  MoveC 565 to (267.87, -55.94, -4.17) mm, rotated rx -180 ry 0 rz -179 deg; joints [20.182, -52.388, 86.98, 32.921, -39.405, -26.577] to (267.42, -56.12, -4.17) mm, rotated rx -180 ry 0 rz -179 deg; joints [20.193, -52.411, 87.018, 32.927, -39.423, -26.576]
  MoveL 566 to (266.79, -56.12, -4.17) mm, rotated rx 180 ry 0 rz -179 deg; joints [20.201, -52.449, 87.082, 32.92, -39.448, -26.562]
  MoveC 567 to (266.34, -56.12, -3.99) mm, rotated rx -180 ry 0 rz -179 deg; joints [20.206, -52.481, 87.122, 32.922, -39.457, -26.561] to (266.15, -56.12, -3.54) mm, rotated rx -180 ry 0 rz -179 deg; joints [20.208, -52.505, 87.128, 32.937, -39.444, -26.579]
  Set speed (500.0 mm/s)
  MoveL 568 to (266.15, -56.12, 5) mm, rotated rx 180 ry 0 rz -179 deg; joints [20.208, -52.749, 86.893, 33.257, -39.042, -26.992]
  MoveL 569 to (266.15, -54.85, 5) mm, rotated rx -180 ry 0 rz -179 deg; joints [20.166, -52.775, 86.937, 33.185, -39.038, -26.93]
  Set speed (25.4 mm/s)
  MoveL 570 to (266.15, -54.85, 1.83) mm, rotated rx -180 ry 0 rz -179 deg; joints [20.166, -52.685, 87.025, 33.065, -39.187, -26.776]
  MoveL 571 to (266.15, -54.85, -7.71) mm, rotated rx -180 ry 0 rz -179 deg; joints [20.166, -52.411, 87.285, 32.712, -39.636, -26.319]
  MoveC 572 to (266.34, -54.85, -8.16) mm, rotated rx -180 ry 0 rz -179 deg; joints [20.164, -52.386, 87.279, 32.698, -39.65, -26.301] to (266.79, -54.85, -8.35) mm, rotated rx -180 ry 0 rz -179 deg; joints [20.158, -52.354, 87.239, 32.696, -39.641, -26.302]
  Set speed (50.8 mm/s)
  MoveL 573 to (267.42, -54.85, -8.35) mm, rotated rx 180 ry 0 rz -179 deg; joints [20.151, -52.317, 87.175, 32.702, -39.616, -26.316]
  MoveC 574 to (267.87, -55.04, -8.35) mm, rotated rx -180 ry 0 rz -179 deg; joints [20.152, -52.286, 87.124, 32.717, -39.599, -26.335] to (268.06, -55.49, -8.35) mm, rotated rx 180 ry 0 rz -179 deg; joints [20.165, -52.266, 87.09, 32.744, -39.593, -26.361]
  MoveL 575 to (268.06, -80.89, -8.35) mm, rotated rx -180 ry 0 rz -179 deg; joints [21.006, -51.73, 86.183, 34.166, -39.665, -27.586]
  MoveL 576 to (217.26, -80.89, -8.35) mm, rotated rx -180 ry 0 rz -179 deg; joints [21.633, -54.688, 91.144, 33.721, -41.611, -26.521]
  MoveL 577 to (217.26, -30.09, -8.35) mm, rotated rx -180 ry 0 rz -179 deg; joints [19.898, -55.732, 92.869, 30.944, -41.444, -24.2]
  MoveL 578 to (268.06, -30.09, -8.35) mm, rotated rx 180 ry 0 rz -179 deg; joints [19.315, -52.777, 87.951, 31.318, -39.52, -25.143]
  MoveL 579 to (268.06, -55.49, -8.35) mm, rotated rx 180 ry 0 rz -179 deg; joints [20.165, -52.266, 87.09, 32.744, -39.593, -26.361]
  MoveC 580 to (267.87, -55.94, -8.35) mm, rotated rx -180 ry 0 rz -179 deg; joints [20.182, -52.268, 87.093, 32.768, -39.601, -26.378] to (267.42, -56.12, -8.35) mm, rotated rx -180 ry 0 rz -179 deg; joints [20.193, -52.291, 87.131, 32.773, -39.62, -26.377]
  MoveL 581 to (266.79, -56.12, -8.35) mm, rotated rx -180 ry 0 rz -179 deg; joints [20.201, -52.328, 87.195, 32.767, -39.645, -26.363]
  MoveC 582 to (266.34, -56.12, -8.16) mm, rotated rx -180 ry 0 rz -179 deg; joints [20.206, -52.36, 87.235, 32.769, -39.654, -26.362] to (266.15, -56.12, -7.72) mm, rotated rx 180 ry 0 rz -179 deg; joints [20.208, -52.384, 87.241, 32.783, -39.64, -26.38]
  Set speed (500.0 mm/s)
  MoveL 583 to (266.15, -56.12, 6) mm, rotated rx -180 ry 0 rz -179 deg; joints [20.208, -52.777, 86.865, 33.295, -38.995, -27.041]
  MoveL 584 to (139.15, -54.85, 6) mm, rotated rx -180 ry 0 rz -179 deg; joints [21.754, -60.075, 98.759, 32.555, -43.53, -24.838]
  Set speed (25.4 mm/s)
  MoveL 585 to (139.15, -54.85, -3.54) mm, rotated rx 180 ry 0 rz -179 deg; joints [21.754, -59.764, 99.016, 32.238, -44.009, -24.398]
  MoveC 586 to (139.34, -54.85, -3.99) mm, rotated rx -180 ry 0 rz -179 deg; joints [21.751, -59.739, 99.012, 32.223, -44.026, -24.38] to (139.79, -54.85, -4.17) mm, rotated rx 180 ry 0 rz -179 deg; joints [21.745, -59.708, 98.977, 32.217, -44.02, -24.377]
  Set speed (50.8 mm/s)
  MoveL 587 to (140.42, -54.85, -4.17) mm, rotated rx -180 ry 0 rz -179 deg; joints [21.736, -59.673, 98.922, 32.217, -43.999, -24.385]
  MoveC 588 to (140.87, -55.04, -4.18) mm, rotated rx -180 ry 0 rz -179 deg; joints [21.737, -59.645, 98.876, 32.227, -43.985, -24.398] to (141.06, -55.49, -4.17) mm, rotated rx 180 ry 0 rz -179 deg; joints [21.75, -59.625, 98.845, 32.251, -43.981, -24.42]
  MoveL 589 to (141.06, -80.89, -4.17) mm, rotated rx 180 ry 0 rz -179 deg; joints [22.648, -59.084, 97.981, 33.603, -44.09, -25.514]
  MoveL 590 to (90.26, -80.89, -4.17) mm, rotated rx -180 ry 0 rz -179 deg; joints [23.379, -61.842, 102.338, 33.653, -45.731, -24.924]
  MoveL 591 to (90.26, -30.09, -4.17) mm, rotated rx -180 ry 0 rz -179 deg; joints [21.523, -62.92, 104.009, 30.966, -45.482, -22.818]
  MoveL 592 to (141.06, -30.09, -4.18) mm, rotated rx 180 ry 0 rz -179 deg; joints [20.842, -60.143, 99.667, 30.888, -43.873, -23.328]
  MoveL 593 to (141.06, -55.49, -4.17) mm, rotated rx 180 ry 0 rz -179 deg; joints [21.75, -59.625, 98.845, 32.251, -43.981, -24.42]
  MoveC 594 to (140.87, -55.94, -4.17) mm, rotated rx -180 ry 0 rz -179 deg; joints [21.769, -59.626, 98.847, 32.275, -43.989, -24.437] to (140.42, -56.12, -4.17) mm, rotated rx -180 ry 0 rz -179 deg; joints [21.782, -59.647, 98.88, 32.285, -44.005, -24.439]
  MoveL 595 to (139.79, -56.12, -4.18) mm, rotated rx -180 ry 0 rz -179 deg; joints [21.79, -59.682, 98.935, 32.285, -44.026, -24.431]
  MoveC 596 to (139.34, -56.12, -3.99) mm, rotated rx 180 ry 0 rz -179 deg; joints [21.796, -59.713, 98.97, 32.291, -44.031, -24.434] to (139.15, -56.12, -3.54) mm, rotated rx -180 ry 0 rz -179 deg; joints [21.799, -59.738, 98.974, 32.305, -44.015, -24.453]
  Set speed (500.0 mm/s)
  MoveL 597 to (139.15, -56.12, 5) mm, rotated rx -180 ry 0 rz -179 deg; joints [21.799, -60.016, 98.744, 32.59, -43.586, -24.847]
  MoveL 598 to (139.15, -54.85, 5) mm, rotated rx -180 ry 0 rz -179 deg; joints [21.754, -60.043, 98.786, 32.522, -43.58, -24.792]
  Set speed (25.4 mm/s)
  MoveL 599 to (139.15, -54.85, 1.83) mm, rotated rx -180 ry 0 rz -179 deg; joints [21.754, -59.94, 98.873, 32.415, -43.74, -24.644]
  MoveL 600 to (139.15, -54.85, -7.72) mm, rotated rx -180 ry 0 rz -179 deg; joints [21.754, -59.626, 99.126, 32.101, -44.219, -24.208]
  MoveC 601 to (139.34, -54.85, -8.16) mm, rotated rx -180 ry 0 rz -179 deg; joints [21.751, -59.601, 99.122, 32.087, -44.236, -24.19] to (139.79, -54.85, -8.35) mm, rotated rx -180 ry 0 rz -179 deg; joints [21.745, -59.57, 99.087, 32.081, -44.23, -24.187]
  Set speed (50.8 mm/s)
  MoveL 602 to (140.42, -54.85, -8.35) mm, rotated rx 180 ry 0 rz -179 deg; joints [21.736, -59.535, 99.032, 32.081, -44.209, -24.195]
  MoveC 603 to (140.87, -55.04, -8.35) mm, rotated rx 180 ry 0 rz -179 deg; joints [21.737, -59.507, 98.986, 32.091, -44.195, -24.209] to (141.06, -55.49, -8.35) mm, rotated rx 180 ry 0 rz -179 deg; joints [21.75, -59.487, 98.955, 32.115, -44.191, -24.23]
  MoveL 604 to (141.06, -80.89, -8.35) mm, rotated rx 180 ry 0 rz -179 deg; joints [22.648, -58.947, 98.091, 33.463, -44.295, -25.318]
  MoveL 605 to (90.26, -80.89, -8.35) mm, rotated rx -180 ry 0 rz -179 deg; joints [23.379, -61.699, 102.448, 33.516, -45.942, -24.728]
  MoveL 606 to (90.26, -30.09, -8.35) mm, rotated rx -180 ry 0 rz -179 deg; joints [21.523, -62.774, 104.119, 30.837, -45.702, -22.634]
  MoveL 607 to (141.06, -30.09, -8.35) mm, rotated rx 180 ry 0 rz -179 deg; joints [20.842, -60.004, 99.777, 30.756, -44.086, -23.144]
  MoveL 608 to (141.06, -55.49, -8.35) mm, rotated rx 180 ry 0 rz -179 deg; joints [21.75, -59.487, 98.955, 32.115, -44.191, -24.23]
  MoveC 609 to (140.87, -55.94, -8.35) mm, rotated rx 180 ry 0 rz -179 deg; joints [21.769, -59.488, 98.956, 32.139, -44.199, -24.247] to (140.42, -56.12, -8.35) mm, rotated rx 180 ry 0 rz -179 deg; joints [21.782, -59.509, 98.99, 32.149, -44.214, -24.249]
  MoveL 610 to (139.79, -56.12, -8.35) mm, rotated rx -180 ry 0 rz -179 deg; joints [21.79, -59.544, 99.045, 32.149, -44.235, -24.242]
  MoveC 611 to (139.34, -56.12, -8.16) mm, rotated rx -180 ry 0 rz -179 deg; joints [21.796, -59.575, 99.08, 32.155, -44.241, -24.245] to (139.15, -56.12, -7.72) mm, rotated rx -180 ry 0 rz -179 deg; joints [21.799, -59.6, 99.084, 32.169, -44.225, -24.263]
  Set speed (500.0 mm/s)
  MoveL 612 to (139.15, -56.12, 6) mm, rotated rx -180 ry 0 rz -179 deg; joints [21.799, -60.049, 98.717, 32.624, -43.536, -24.893]
  MoveL 613 to (139.15, -235.88, 6) mm, rotated rx -180 ry 0 rz -179 deg; joints [27.912, -55.671, 91.665, 42.031, -44.36, -32.8]
  Set speed (25.4 mm/s)
  MoveL 614 to (139.15, -235.88, -3.54) mm, rotated rx -180 ry 0 rz -179 deg; joints [27.912, -55.384, 91.924, 41.661, -44.767, -32.28]
  MoveC 615 to (139.34, -235.88, -3.99) mm, rotated rx -180 ry 0 rz -179 deg; joints [27.909, -55.36, 91.92, 41.644, -44.78, -32.26] to (139.79, -235.88, -4.17) mm, rotated rx 180 ry 0 rz -179 deg; joints [27.902, -55.33, 91.885, 41.639, -44.772, -32.258]
  Set speed (50.8 mm/s)
  MoveL 616 to (140.42, -235.89, -4.17) mm, rotated rx -180 ry 0 rz -179 deg; joints [27.891, -55.296, 91.828, 41.641, -44.75, -32.27]
  MoveC 617 to (140.87, -236.07, -4.18) mm, rotated rx 180 ry 0 rz -179 deg; joints [27.89, -55.266, 91.779, 41.653, -44.735, -32.287] to (141.06, -236.52, -4.17) mm, rotated rx 180 ry 0 rz -179 deg; joints [27.901, -55.244, 91.742, 41.676, -44.73, -32.311]
  MoveL 618 to (141.06, -261.92, -4.17) mm, rotated rx -180 ry 0 rz -179 deg; joints [28.717, -54.531, 90.562, 42.965, -44.828, -33.447]
  MoveL 619 to (90.26, -261.92, -4.17) mm, rotated rx 180 ry 0 rz -179 deg; joints [29.592, -57.246, 95.019, 42.834, -46.58, -32.507]
  MoveL 620 to (90.26, -211.12, -4.17) mm, rotated rx -180 ry 0 rz -179 deg; joints [27.914, -58.655, 97.294, 40.313, -46.353, -30.353]
  MoveL 621 to (141.06, -211.12, -4.17) mm, rotated rx -180 ry 0 rz -179 deg; joints [27.074, -55.932, 92.875, 40.38, -44.63, -31.184]
  MoveL 622 to (141.06, -236.52, -4.17) mm, rotated rx -180 ry 0 rz -179 deg; joints [27.901, -55.244, 91.742, 41.676, -44.73, -32.311]
  MoveC 623 to (140.87, -236.97, -4.18) mm, rotated rx -180 ry 0 rz -179 deg; joints [27.919, -55.241, 91.738, 41.698, -44.738, -32.327] to (140.42, -237.15, -4.18) mm, rotated rx 180 ry 0 rz -179 deg; joints [27.932, -55.261, 91.77, 41.706, -44.755, -32.327]
  MoveL 624 to (139.79, -237.15, -4.18) mm, rotated rx -180 ry 0 rz -179 deg; joints [27.943, -55.295, 91.827, 41.703, -44.777, -32.315]
  MoveC 625 to (139.34, -237.16, -3.99) mm, rotated rx -180 ry 0 rz -179 deg; joints [27.95, -55.325, 91.862, 41.709, -44.785, -32.316] to (139.15, -237.15, -3.54) mm, rotated rx -180 ry 0 rz -179 deg; joints [27.953, -55.349, 91.867, 41.725, -44.772, -32.337]
  Set speed (500.0 mm/s)
  MoveL 626 to (139.15, -237.15, 5) mm, rotated rx -180 ry 0 rz -179 deg; joints [27.953, -55.606, 91.635, 42.057, -44.408, -32.802]
  MoveL 627 to (139.15, -235.88, 5) mm, rotated rx -180 ry 0 rz -179 deg; joints [27.912, -55.641, 91.693, 41.992, -44.403, -32.745]
  Set speed (25.4 mm/s)
  MoveL 628 to (139.15, -235.88, 1.83) mm, rotated rx -180 ry 0 rz -179 deg; joints [27.912, -55.546, 91.779, 41.868, -44.538, -32.571]
  MoveL 629 to (139.15, -235.88, -7.72) mm, rotated rx 180 ry 0 rz -179 deg; joints [27.912, -55.257, 92.036, 41.502, -44.946, -32.056]
  MoveC 630 to (139.34, -235.88, -8.16) mm, rotated rx -180 ry 0 rz -179 deg; joints [27.909, -55.233, 92.031, 41.485, -44.959, -32.035] to (139.79, -235.88, -8.35) mm, rotated rx 180 ry 0 rz -179 deg; joints [27.902, -55.203, 91.996, 41.48, -44.951, -32.034]
  Set speed (50.8 mm/s)
  MoveL 631 to (140.42, -235.89, -8.35) mm, rotated rx -180 ry 0 rz -179 deg; joints [27.891, -55.168, 91.939, 41.482, -44.928, -32.046]
  MoveC 632 to (140.87, -236.07, -8.35) mm, rotated rx -180 ry 0 rz -179 deg; joints [27.89, -55.139, 91.89, 41.493, -44.913, -32.063] to (141.06, -236.52, -8.35) mm, rotated rx -180 ry 0 rz -179 deg; joints [27.901, -55.116, 91.853, 41.517, -44.908, -32.087]
  MoveL 633 to (141.06, -261.92, -8.35) mm, rotated rx -180 ry 0 rz -179 deg; joints [28.717, -54.405, 90.673, 42.803, -45.001, -33.219]
  MoveL 634 to (90.26, -261.92, -8.35) mm, rotated rx -180 ry 0 rz -179 deg; joints [29.592, -57.114, 95.129, 42.679, -46.758, -32.28]
  MoveL 635 to (90.26, -211.12, -8.35) mm, rotated rx -180 ry 0 rz -179 deg; joints [27.914, -58.519, 97.404, 40.162, -46.54, -30.135]
  MoveL 636 to (141.06, -211.12, -8.35) mm, rotated rx -180 ry 0 rz -179 deg; joints [27.074, -55.803, 92.986, 40.224, -44.813, -30.964]
  MoveL 637 to (141.06, -236.52, -8.35) mm, rotated rx -180 ry 0 rz -179 deg; joints [27.901, -55.116, 91.853, 41.517, -44.908, -32.087]
  MoveC 638 to (140.87, -236.97, -8.35) mm, rotated rx -180 ry 0 rz -179 deg; joints [27.919, -55.114, 91.849, 41.539, -44.916, -32.103] to (140.42, -237.16, -8.35) mm, rotated rx -180 ry 0 rz -179 deg; joints [27.932, -55.133, 91.881, 41.547, -44.933, -32.102]
  MoveL 639 to (139.79, -237.16, -8.35) mm, rotated rx -180 ry 0 rz -179 deg; joints [27.943, -55.168, 91.938, 41.544, -44.955, -32.09]
  MoveC 640 to (139.34, -237.15, -8.16) mm, rotated rx 180 ry 0 rz -179 deg; joints [27.95, -55.198, 91.973, 41.55, -44.963, -32.091] to (139.15, -237.15, -7.72) mm, rotated rx -180 ry 0 rz -179 deg; joints [27.953, -55.222, 91.978, 41.566, -44.951, -32.112]
  Set speed (500.0 mm/s)
  MoveL 641 to (139.15, -237.15, 6) mm, rotated rx -180 ry 0 rz -179 deg; joints [27.953, -55.636, 91.607, 42.096, -44.366, -32.857]
  MoveL 642 to (266.15, -235.88, 6) mm, rotated rx -180 ry 0 rz -179 deg; joints [25.965, -48.371, 79.367, 43.399, -39.586, -36.084]
  Set speed (25.4 mm/s)
  MoveL 643 to (266.15, -235.89, -3.54) mm, rotated rx -180 ry 0 rz -179 deg; joints [25.965, -48.122, 79.642, 42.969, -39.967, -35.524]
  MoveC 644 to (266.34, -235.88, -3.99) mm, rotated rx -180 ry 0 rz -179 deg; joints [25.963, -48.099, 79.635, 42.953, -39.977, -35.504] to (266.79, -235.89, -4.17) mm, rotated rx -180 ry 0 rz -179 deg; joints [25.956, -48.067, 79.593, 42.953, -39.966, -35.509]
  Set speed (50.8 mm/s)
  MoveL 645 to (267.42, -235.89, -4.18) mm, rotated rx -180 ry 0 rz -179 deg; joints [25.947, -48.029, 79.526, 42.964, -39.94, -35.53]
  MoveC 646 to (267.87, -236.07, -4.17) mm, rotated rx 180 ry 0 rz -179 deg; joints [25.947, -47.996, 79.47, 42.983, -39.923, -35.554] to (268.06, -236.52, -4.18) mm, rotated rx -180 ry 0 rz -179 deg; joints [25.958, -47.972, 79.428, 43.011, -39.916, -35.584]
  MoveL 647 to (268.06, -261.92, -4.18) mm, rotated rx 180 ry 0 rz -179 deg; joints [26.731, -47.239, 78.154, 44.43, -39.983, -36.912]
  MoveL 648 to (217.26, -261.92, -4.18) mm, rotated rx -180 ry 0 rz -179 deg; joints [27.493, -50.26, 83.367, 43.615, -42.008, -35.297]
  MoveL 649 to (217.26, -211.12, -4.17) mm, rotated rx -180 ry 0 rz -179 deg; joints [25.902, -51.672, 85.769, 40.9, -41.85, -32.832]
  MoveL 650 to (268.06, -211.12, -4.17) mm, rotated rx 180 ry 0 rz -179 deg; joints [25.174, -48.676, 80.646, 41.595, -39.848, -34.275]
  MoveL 651 to (268.06, -236.52, -4.18) mm, rotated rx -180 ry 0 rz -179 deg; joints [25.958, -47.972, 79.428, 43.011, -39.916, -35.584]
  MoveC 652 to (267.87, -236.97, -4.17) mm, rotated rx -180 ry 0 rz -179 deg; joints [25.974, -47.971, 79.426, 43.033, -39.925, -35.601] to (267.42, -237.16, -4.18) mm, rotated rx 180 ry 0 rz -179 deg; joints [25.986, -47.993, 79.464, 43.035, -39.944, -35.596]
  MoveL 653 to (266.79, -237.15, -4.17) mm, rotated rx -180 ry 0 rz -179 deg; joints [25.995, -48.031, 79.531, 43.023, -39.97, -35.574]
  MoveC 654 to (266.34, -237.15, -3.99) mm, rotated rx 180 ry 0 rz -179 deg; joints [26.002, -48.063, 79.573, 43.024, -39.981, -35.57] to (266.15, -237.16, -3.54) mm, rotated rx -180 ry 0 rz -179 deg; joints [26.004, -48.087, 79.579, 43.04, -39.97, -35.59]
  Set speed (500.0 mm/s)
  MoveL 655 to (266.15, -237.15, 5) mm, rotated rx 180 ry 0 rz -179 deg; joints [26.004, -48.309, 79.334, 43.425, -39.629, -36.091]
  MoveL 656 to (266.15, -235.89, 5) mm, rotated rx -180 ry 0 rz -179 deg; joints [25.965, -48.345, 79.397, 43.354, -39.626, -36.024]
  Set speed (25.4 mm/s)
  MoveL 657 to (266.15, -235.88, 1.83) mm, rotated rx 180 ry 0 rz -179 deg; joints [25.965, -48.263, 79.488, 43.21, -39.752, -35.837]
  MoveL 658 to (266.15, -235.89, -7.71) mm, rotated rx -180 ry 0 rz -179 deg; joints [25.965, -48.012, 79.759, 42.785, -40.134, -35.283]
  MoveC 659 to (266.34, -235.88, -8.16) mm, rotated rx 180 ry 0 rz -179 deg; joints [25.963, -47.989, 79.752, 42.769, -40.144, -35.264] to (266.79, -235.89, -8.35) mm, rotated rx -180 ry 0 rz -179 deg; joints [25.956, -47.957, 79.71, 42.768, -40.133, -35.268]
  Set speed (50.8 mm/s)
  MoveL 660 to (267.42, -235.89, -8.35) mm, rotated rx -180 ry 0 rz -179 deg; joints [25.947, -47.918, 79.643, 42.78, -40.107, -35.289]
  MoveC 661 to (267.87, -236.07, -8.35) mm, rotated rx -180 ry 0 rz -179 deg; joints [25.947, -47.886, 79.587, 42.798, -40.089, -35.313] to (268.06, -236.52, -8.35) mm, rotated rx -180 ry 0 rz -179 deg; joints [25.958, -47.862, 79.545, 42.826, -40.083, -35.343]
  MoveL 662 to (268.06, -261.92, -8.35) mm, rotated rx -180 ry 0 rz -179 deg; joints [26.731, -47.13, 78.272, 44.241, -40.145, -36.665]
  MoveL 663 to (217.26, -261.92, -8.35) mm, rotated rx -180 ry 0 rz -179 deg; joints [27.493, -50.144, 83.481, 43.439, -42.175, -35.06]
  MoveL 664 to (217.26, -211.12, -8.35) mm, rotated rx -180 ry 0 rz -179 deg; joints [25.902, -51.553, 85.883, 40.731, -42.026, -32.605]
  MoveL 665 to (268.06, -211.12, -8.35) mm, rotated rx 180 ry 0 rz -179 deg; joints [25.174, -48.564, 80.762, 41.414, -40.019, -34.04]
  MoveL 666 to (268.06, -236.52, -8.35) mm, rotated rx -180 ry 0 rz -179 deg; joints [25.958, -47.862, 79.545, 42.826, -40.083, -35.343]
  MoveC 667 to (267.87, -236.97, -8.35) mm, rotated rx -180 ry 0 rz -179 deg; joints [25.974, -47.86, 79.543, 42.848, -40.092, -35.36] to (267.42, -237.16, -8.35) mm, rotated rx -180 ry 0 rz -179 deg; joints [25.986, -47.882, 79.581, 42.85, -40.11, -35.354]
  MoveL 668 to (266.79, -237.15, -8.35) mm, rotated rx -180 ry 0 rz -179 deg; joints [25.995, -47.921, 79.648, 42.839, -40.136, -35.333]
  MoveC 669 to (266.34, -237.15, -8.16) mm, rotated rx 180 ry 0 rz -179 deg; joints [26.002, -47.953, 79.69, 42.839, -40.147, -35.329] to (266.15, -237.16, -7.72) mm, rotated rx -180 ry 0 rz -179 deg; joints [26.004, -47.976, 79.697, 42.856, -40.137, -35.349]
  Set speed (500.0 mm/s)
  MoveL 670 to (266.15, -237.16, 6) mm, rotated rx -180 ry 0 rz -179 deg; joints [26.004, -48.335, 79.305, 43.471, -39.59, -36.15]
  MoveL 671 to (393.15, -235.88, 6) mm, rotated rx -180 ry 0 rz -179 deg; joints [24.267, -39.923, 64.425, 47.387, -33.948, -42.041]
  Set speed (25.4 mm/s)
  MoveL 672 to (393.15, -235.88, -3.54) mm, rotated rx -180 ry 0 rz -179 deg; joints [24.267, -39.722, 64.741, 46.829, -34.299, -41.367]
  MoveC 673 to (393.34, -235.88, -3.99) mm, rotated rx 180 ry 0 rz -179 deg; joints [24.264, -39.699, 64.731, 46.812, -34.307, -41.348] to (393.79, -235.89, -4.17) mm, rotated rx -180 ry 0 rz -179 deg; joints [24.259, -39.662, 64.677, 46.822, -34.292, -41.363]
  Set speed (50.8 mm/s)
  MoveL 674 to (394.42, -235.88, -4.18) mm, rotated rx 180 ry 0 rz -179 deg; joints [24.251, -39.615, 64.592, 46.852, -34.26, -41.404]
  MoveC 675 to (394.87, -236.07, -4.18) mm, rotated rx -180 ry 0 rz -179 deg; joints [24.25, -39.576, 64.522, 46.886, -34.239, -41.445] to (395.06, -236.52, -4.17) mm, rotated rx -180 ry 0 rz -179 deg; joints [24.261, -39.549, 64.471, 46.925, -34.23, -41.486]
  MoveL 676 to (395.06, -261.92, -4.18) mm, rotated rx -180 ry 0 rz -179 deg; joints [24.996, -38.724, 62.973, 48.623, -34.272, -43.171]
  MoveL 677 to (344.26, -261.92, -4.18) mm, rotated rx 180 ry 0 rz -179 deg; joints [25.663, -42.34, 69.501, 46.465, -36.682, -40.167]
  MoveL 678 to (344.26, -211.12, -4.17) mm, rotated rx -180 ry 0 rz -179 deg; joints [24.154, -43.854, 72.2, 43.366, -36.579, -37.18]
  MoveL 679 to (395.06, -211.12, -4.18) mm, rotated rx 180 ry 0 rz -179 deg; joints [23.519, -40.332, 65.889, 45.25, -34.187, -39.843]
  MoveL 680 to (395.06, -236.52, -4.17) mm, rotated rx -180 ry 0 rz -179 deg; joints [24.261, -39.549, 64.471, 46.925, -34.23, -41.486]
  MoveC 681 to (394.87, -236.97, -4.18) mm, rotated rx 180 ry 0 rz -179 deg; joints [24.277, -39.548, 64.47, 46.946, -34.24, -41.503] to (394.42, -237.16, -4.18) mm, rotated rx 180 ry 0 rz -179 deg; joints [24.288, -39.575, 64.52, 46.937, -34.263, -41.487]
  MoveL 682 to (393.79, -237.16, -4.17) mm, rotated rx -180 ry 0 rz -179 deg; joints [24.296, -39.622, 64.604, 46.907, -34.294, -41.446]
  MoveC 683 to (393.34, -237.15, -3.99) mm, rotated rx -180 ry 0 rz -179 deg; joints [24.301, -39.659, 64.658, 46.896, -34.309, -41.431] to (393.15, -237.16, -3.54) mm, rotated rx 180 ry 0 rz -179 deg; joints [24.304, -39.682, 64.668, 46.913, -34.302, -41.45]
  Set speed (500.0 mm/s)
  MoveL 684 to (393.15, -237.16, 5) mm, rotated rx -180 ry 0 rz -179 deg; joints [24.304, -39.862, 64.386, 47.412, -33.988, -42.054]
  MoveL 685 to (393.15, -235.88, 5) mm, rotated rx -180 ry 0 rz -179 deg; joints [24.267, -39.902, 64.459, 47.328, -33.985, -41.97]
  Set speed (25.4 mm/s)
  MoveL 686 to (393.15, -235.88, 1.82) mm, rotated rx 180 ry 0 rz -179 deg; joints [24.267, -39.836, 64.565, 47.141, -34.102, -41.744]
  MoveL 687 to (393.15, -235.88, -7.72) mm, rotated rx -180 ry 0 rz -179 deg; joints [24.267, -39.632, 64.875, 46.59, -34.453, -41.078]
  MoveC 688 to (393.34, -235.88, -8.16) mm, rotated rx 180 ry 0 rz -179 deg; joints [24.264, -39.609, 64.865, 46.573, -34.461, -41.059] to (393.79, -235.89, -8.35) mm, rotated rx 180 ry 0 rz -179 deg; joints [24.259, -39.572, 64.811, 46.584, -34.446, -41.074]
  Set speed (50.8 mm/s)
  MoveL 689 to (394.42, -235.89, -8.35) mm, rotated rx -180 ry 0 rz -179 deg; joints [24.251, -39.526, 64.727, 46.613, -34.414, -41.114]
  MoveC 690 to (394.87, -236.07, -8.35) mm, rotated rx -180 ry 0 rz -179 deg; joints [24.25, -39.487, 64.657, 46.647, -34.392, -41.155] to (395.06, -236.52, -8.35) mm, rotated rx -180 ry 0 rz -179 deg; joints [24.261, -39.459, 64.606, 46.685, -34.384, -41.196]
  MoveL 691 to (395.06, -261.92, -8.35) mm, rotated rx -180 ry 0 rz -179 deg; joints [24.996, -38.637, 63.11, 48.377, -34.421, -42.872]
  MoveL 692 to (344.26, -261.92, -8.35) mm, rotated rx -180 ry 0 rz -179 deg; joints [25.663, -42.243, 69.629, 46.248, -36.837, -39.896]
  MoveL 693 to (344.26, -211.12, -8.35) mm, rotated rx 180 ry 0 rz -179 deg; joints [24.154, -43.753, 72.324, 43.159, -36.742, -36.922]
  MoveL 694 to (395.06, -211.12, -8.35) mm, rotated rx -180 ry 0 rz -179 deg; joints [23.519, -40.24, 66.022, 45.016, -34.345, -39.561]
  MoveL 695 to (395.06, -236.52, -8.35) mm, rotated rx -180 ry 0 rz -179 deg; joints [24.261, -39.459, 64.606, 46.685, -34.384, -41.196]
  MoveC 696 to (394.87, -236.97, -8.35) mm, rotated rx -180 ry 0 rz -179 deg; joints [24.277, -39.459, 64.605, 46.706, -34.394, -41.213] to (394.42, -237.16, -8.35) mm, rotated rx -180 ry 0 rz -179 deg; joints [24.288, -39.486, 64.654, 46.697, -34.416, -41.197]
  MoveL 697 to (393.79, -237.16, -8.35) mm, rotated rx -180 ry 0 rz -179 deg; joints [24.296, -39.532, 64.739, 46.667, -34.447, -41.157]
  MoveC 698 to (393.34, -237.15, -8.16) mm, rotated rx -180 ry 0 rz -179 deg; joints [24.301, -39.569, 64.793, 46.657, -34.463, -41.141] to (393.15, -237.16, -7.72) mm, rotated rx -180 ry 0 rz -179 deg; joints [24.304, -39.592, 64.803, 46.674, -34.455, -41.16]
  Set speed (500.0 mm/s)
  MoveL 699 to (393.15, -237.16, 6) mm, rotated rx -180 ry 0 rz -179 deg; joints [24.304, -39.882, 64.352, 47.472, -33.951, -42.125]
  MoveL 700 to (393.15, -422.22, 6) mm, rotated rx 180 ry 0 rz -179 deg; joints [29.464, -32.65, 51.048, 60.809, -34.294, -55.932]
  Set speed (25.4 mm/s)
  MoveL 701 to (393.15, -422.22, -3.54) mm, rotated rx -180 ry 0 rz -179 deg; joints [29.464, -32.503, 51.438, 60.128, -34.558, -55.107]
  MoveC 702 to (393.34, -422.22, -3.99) mm, rotated rx -180 ry 0 rz -179 deg; joints [29.462, -32.479, 51.425, 60.112, -34.562, -55.088] to (393.79, -422.22, -4.17) mm, rotated rx 180 ry 0 rz -179 deg; joints [29.455, -32.437, 51.358, 60.136, -34.544, -55.12]
  Set speed (50.8 mm/s)
  MoveL 703 to (394.42, -422.22, -4.18) mm, rotated rx 180 ry 0 rz -179 deg; joints [29.446, -32.38, 51.252, 60.189, -34.512, -55.187]
  MoveC 704 to (394.87, -422.41, -4.17) mm, rotated rx -180 ry 0 rz -179 deg; joints [29.445, -32.331, 51.161, 60.241, -34.49, -55.252] to (395.06, -422.86, -4.17) mm, rotated rx -180 ry 0 rz -179 deg; joints [29.454, -32.293, 51.089, 60.293, -34.481, -55.311]
  MoveL 705 to (395.06, -448.26, -4.17) mm, rotated rx -180 ry 0 rz -179 deg; joints [30.126, -31.02, 48.698, 62.376, -34.505, -57.583]
  MoveL 706 to (344.26, -448.26, -4.17) mm, rotated rx -180 ry 0 rz -179 deg; joints [30.888, -35.354, 56.786, 58.582, -36.981, -52.597]
  MoveL 707 to (344.26, -397.46, -4.17) mm, rotated rx -180 ry 0 rz -179 deg; joints [29.512, -37.525, 60.781, 55.102, -36.914, -48.897]
  MoveL 708 to (395.06, -397.46, -4.18) mm, rotated rx -180 ry 0 rz -179 deg; joints [28.773, -33.479, 53.306, 58.299, -34.454, -53.166]
  MoveL 709 to (395.06, -422.86, -4.17) mm, rotated rx -180 ry 0 rz -179 deg; joints [29.454, -32.293, 51.089, 60.293, -34.481, -55.311]
  MoveC 710 to (394.87, -423.31, -4.18) mm, rotated rx 180 ry 0 rz -179 deg; joints [29.469, -32.288, 51.08, 60.313, -34.491, -55.329] to (394.42, -423.49, -4.18) mm, rotated rx 180 ry 0 rz -179 deg; joints [29.48, -32.319, 51.138, 60.29, -34.513, -55.297]
  MoveL 711 to (393.79, -423.49, -4.18) mm, rotated rx -180 ry 0 rz -179 deg; joints [29.489, -32.376, 51.244, 60.237, -34.545, -55.23]
  MoveC 712 to (393.34, -423.49, -3.99) mm, rotated rx -180 ry 0 rz -179 deg; joints [29.496, -32.418, 51.311, 60.213, -34.563, -55.198] to (393.15, -423.49, -3.54) mm, rotated rx 180 ry 0 rz -179 deg; joints [29.498, -32.442, 51.324, 60.229, -34.56, -55.216]
  Set speed (500.0 mm/s)
  MoveL 713 to (393.15, -423.49, 5) mm, rotated rx -180 ry 0 rz -179 deg; joints [29.498, -32.573, 50.974, 60.839, -34.324, -55.955]
  MoveL 714 to (393.15, -422.22, 5) mm, rotated rx 180 ry 0 rz -179 deg; joints [29.464, -32.635, 51.09, 60.737, -34.322, -55.845]
  Set speed (25.4 mm/s)
  MoveL 715 to (393.15, -422.22, 1.82) mm, rotated rx -180 ry 0 rz -179 deg; joints [29.464, -32.586, 51.22, 60.509, -34.41, -55.568]
  MoveL 716 to (393.15, -422.22, -7.72) mm, rotated rx 180 ry 0 rz -179 deg; joints [29.464, -32.436, 51.604, 59.836, -34.675, -54.752]
  MoveC 717 to (393.34, -422.22, -8.16) mm, rotated rx 180 ry 0 rz -179 deg; joints [29.462, -32.413, 51.591, 59.82, -34.678, -54.734] to (393.79, -422.22, -8.35) mm, rotated rx -180 ry 0 rz -179 deg; joints [29.455, -32.37, 51.524, 59.844, -34.661, -54.765]
  Set speed (50.8 mm/s)
  MoveL 718 to (394.42, -422.22, -8.35) mm, rotated rx -180 ry 0 rz -179 deg; joints [29.446, -32.314, 51.419, 59.896, -34.629, -54.832]
  MoveC 719 to (394.87, -422.41, -8.35) mm, rotated rx -180 ry 0 rz -179 deg; joints [29.445, -32.265, 51.328, 59.948, -34.606, -54.896] to (395.06, -422.86, -8.35) mm, rotated rx -180 ry 0 rz -179 deg; joints [29.454, -32.227, 51.256, 59.999, -34.597, -54.954]
  MoveL 720 to (395.06, -448.26, -8.35) mm, rotated rx -180 ry 0 rz -179 deg; joints [30.126, -30.959, 48.874, 62.073, -34.615, -57.215]
  MoveL 721 to (344.26, -448.26, -8.35) mm, rotated rx 180 ry 0 rz -179 deg; joints [30.888, -35.277, 56.936, 58.325, -37.1, -52.274]
  MoveL 722 to (344.26, -397.46, -8.35) mm, rotated rx -180 ry 0 rz -179 deg; joints [29.512, -37.441, 60.923, 54.857, -37.043, -48.59]
  MoveL 723 to (395.06, -397.46, -8.35) mm, rotated rx 180 ry 0 rz -179 deg; joints [28.773, -33.409, 53.466, 58.014, -34.576, -52.82]
  MoveL 724 to (395.06, -422.86, -8.35) mm, rotated rx -180 ry 0 rz -179 deg; joints [29.454, -32.227, 51.256, 59.999, -34.597, -54.954]
  MoveC 725 to (394.87, -423.31, -8.35) mm, rotated rx 180 ry 0 rz -179 deg; joints [29.469, -32.222, 51.247, 60.019, -34.607, -54.973] to (394.42, -423.49, -8.35) mm, rotated rx -180 ry 0 rz -179 deg; joints [29.48, -32.253, 51.305, 59.997, -34.629, -54.941]
  MoveL 726 to (393.79, -423.49, -8.35) mm, rotated rx -180 ry 0 rz -179 deg; joints [29.489, -32.309, 51.41, 59.945, -34.662, -54.874]
  MoveC 727 to (393.34, -423.49, -8.16) mm, rotated rx 180 ry 0 rz -179 deg; joints [29.496, -32.352, 51.477, 59.921, -34.679, -54.842] to (393.15, -423.49, -7.72) mm, rotated rx 180 ry 0 rz -179 deg; joints [29.498, -32.376, 51.49, 59.937, -34.676, -54.861]
  Set speed (500.0 mm/s)
  MoveL 728 to (393.15, -423.49, 6) mm, rotated rx -180 ry 0 rz -179 deg; joints [29.498, -32.588, 50.933, 60.911, -34.296, -56.043]
  MoveL 729 to (266.15, -422.22, 6) mm, rotated rx 180 ry 0 rz -179 deg; joints [31.414, -42.203, 68.526, 54.019, -40.099, -46.494]
  Set speed (25.4 mm/s)
  MoveL 730 to (266.15, -422.22, -3.54) mm, rotated rx 180 ry 0 rz -179 deg; joints [31.414, -41.989, 68.827, 53.528, -40.404, -45.851]
  MoveC 731 to (266.34, -422.22, -3.99) mm, rotated rx -180 ry 0 rz -179 deg; joints [31.411, -41.966, 68.819, 53.511, -40.41, -45.83] to (266.79, -422.22, -4.17) mm, rotated rx -180 ry 0 rz -179 deg; joints [31.404, -41.933, 68.773, 53.515, -40.397, -45.84]
  Set speed (50.8 mm/s)
  MoveL 732 to (267.42, -422.22, -4.17) mm, rotated rx -180 ry 0 rz -179 deg; joints [31.394, -41.892, 68.698, 53.535, -40.37, -45.873]
  MoveC 733 to (267.87, -422.41, -4.18) mm, rotated rx -180 ry 0 rz -179 deg; joints [31.392, -41.855, 68.633, 53.56, -40.352, -45.907] to (268.06, -422.86, -4.18) mm, rotated rx -180 ry 0 rz -179 deg; joints [31.401, -41.826, 68.581, 53.592, -40.345, -45.943]
  MoveL 734 to (268.06, -448.26, -4.17) mm, rotated rx 180 ry 0 rz -179 deg; joints [32.101, -40.832, 66.792, 55.092, -40.391, -47.504]
  MoveL 735 to (217.26, -448.26, -4.17) mm, rotated rx -180 ry 0 rz -179 deg; joints [32.96, -44.063, 72.571, 53.644, -42.497, -45.048]
  MoveL 736 to (217.26, -397.46, -4.18) mm, rotated rx 180 ry 0 rz -179 deg; joints [31.527, -45.926, 75.859, 50.875, -42.38, -42.245]
  MoveL 737 to (268.06, -397.46, -4.18) mm, rotated rx -180 ry 0 rz -179 deg; joints [30.691, -42.778, 70.284, 52.113, -40.295, -44.428]
  MoveL 738 to (268.06, -422.86, -4.18) mm, rotated rx -180 ry 0 rz -179 deg; joints [31.401, -41.826, 68.581, 53.592, -40.345, -45.943]
  MoveC 739 to (267.87, -423.31, -4.17) mm, rotated rx -180 ry 0 rz -179 deg; joints [31.417, -41.821, 68.571, 53.613, -40.353, -45.961] to (267.42, -423.49, -4.17) mm, rotated rx -180 ry 0 rz -179 deg; joints [31.429, -41.843, 68.611, 53.61, -40.373, -45.949]
  MoveL 740 to (266.79, -423.49, -4.17) mm, rotated rx -180 ry 0 rz -179 deg; joints [31.439, -41.884, 68.685, 53.59, -40.4, -45.917]
  MoveC 741 to (266.34, -423.49, -3.99) mm, rotated rx -180 ry 0 rz -179 deg; joints [31.447, -41.918, 68.732, 53.585, -40.413, -45.907] to (266.15, -423.49, -3.54) mm, rotated rx -180 ry 0 rz -179 deg; joints [31.45, -41.94, 68.74, 53.602, -40.406, -45.927]
  Set speed (500.0 mm/s)
  MoveL 742 to (266.15, -423.49, 5) mm, rotated rx -180 ry 0 rz -179 deg; joints [31.45, -42.132, 68.471, 54.041, -40.134, -46.503]
  MoveL 743 to (266.15, -422.22, 5) mm, rotated rx 180 ry 0 rz -179 deg; joints [31.414, -42.181, 68.558, 53.967, -40.131, -46.426]
  Set speed (25.4 mm/s)
  MoveL 744 to (266.15, -422.22, 1.82) mm, rotated rx 180 ry 0 rz -179 deg; joints [31.414, -42.11, 68.659, 53.802, -40.233, -46.211]
  MoveL 745 to (266.15, -422.22, -7.71) mm, rotated rx -180 ry 0 rz -179 deg; joints [31.414, -41.893, 68.956, 53.317, -40.538, -45.573]
  MoveC 746 to (266.34, -422.22, -8.16) mm, rotated rx 180 ry 0 rz -179 deg; joints [31.411, -41.871, 68.948, 53.3, -40.544, -45.553] to (266.79, -422.22, -8.35) mm, rotated rx 180 ry 0 rz -179 deg; joints [31.404, -41.837, 68.901, 53.304, -40.531, -45.563]
  Set speed (50.8 mm/s)
  MoveL 747 to (267.42, -422.22, -8.35) mm, rotated rx -180 ry 0 rz -179 deg; joints [31.394, -41.796, 68.827, 53.324, -40.504, -45.595]
  MoveC 748 to (267.87, -422.41, -8.35) mm, rotated rx -180 ry 0 rz -179 deg; joints [31.392, -41.76, 68.762, 53.349, -40.485, -45.629] to (268.06, -422.86, -8.35) mm, rotated rx -180 ry 0 rz -179 deg; joints [31.401, -41.73, 68.709, 53.381, -40.478, -45.666]
  MoveL 749 to (268.06, -448.26, -8.35) mm, rotated rx -180 ry 0 rz -179 deg; joints [32.101, -40.739, 66.923, 54.877, -40.52, -47.221]
  MoveL 750 to (217.26, -448.26, -8.35) mm, rotated rx -180 ry 0 rz -179 deg; joints [32.96, -43.962, 72.695, 53.447, -42.63, -44.781]
  MoveL 751 to (217.26, -397.46, -8.35) mm, rotated rx -180 ry 0 rz -179 deg; joints [31.527, -45.821, 75.979, 50.684, -42.522, -41.985]
  MoveL 752 to (268.06, -397.46, -8.35) mm, rotated rx 180 ry 0 rz -179 deg; joints [30.691, -42.68, 70.411, 51.905, -40.433, -44.155]
  MoveL 753 to (268.06, -422.86, -8.35) mm, rotated rx -180 ry 0 rz -179 deg; joints [31.401, -41.73, 68.709, 53.381, -40.478, -45.666]
  MoveC 754 to (267.87, -423.31, -8.35) mm, rotated rx -180 ry 0 rz -179 deg; joints [31.417, -41.725, 68.7, 53.401, -40.487, -45.683] to (267.42, -423.49, -8.35) mm, rotated rx -180 ry 0 rz -179 deg; joints [31.429, -41.747, 68.74, 53.398, -40.506, -45.672]
  MoveL 755 to (266.79, -423.49, -8.35) mm, rotated rx 180 ry 0 rz -179 deg; joints [31.439, -41.789, 68.814, 53.378, -40.533, -45.639]
  MoveC 756 to (266.34, -423.49, -8.16) mm, rotated rx 180 ry 0 rz -179 deg; joints [31.447, -41.822, 68.861, 53.374, -40.546, -45.629] to (266.15, -423.49, -7.72) mm, rotated rx -180 ry 0 rz -179 deg; joints [31.45, -41.845, 68.869, 53.391, -40.54, -45.649]
  Set speed (500.0 mm/s)
  MoveL 757 to (266.15, -423.49, 6) mm, rotated rx 180 ry 0 rz -179 deg; joints [31.45, -42.154, 68.439, 54.093, -40.102, -46.571]
  MoveL 758 to (139.15, -422.22, 6) mm, rotated rx -180 ry 0 rz -179 deg; joints [33.62, -49.808, 81.836, 51.423, -45.092, -41.512]
  Set speed (25.4 mm/s)
  MoveL 759 to (139.15, -422.22, -3.54) mm, rotated rx -180 ry 0 rz -179 deg; joints [33.62, -49.551, 82.106, 51.017, -45.421, -40.934]
  MoveC 760 to (139.34, -422.22, -3.99) mm, rotated rx -180 ry 0 rz -179 deg; joints [33.617, -49.529, 82.101, 51, -45.43, -40.913] to (139.79, -422.22, -4.17) mm, rotated rx 180 ry 0 rz -179 deg; joints [33.608, -49.499, 82.064, 50.997, -45.42, -40.915]
  Set speed (50.8 mm/s)
  MoveL 761 to (140.42, -422.22, -4.18) mm, rotated rx -180 ry 0 rz -179 deg; joints [33.597, -49.464, 82.003, 51.004, -45.396, -40.934]
  MoveC 762 to (140.87, -422.41, -4.17) mm, rotated rx 180 ry 0 rz -179 deg; joints [33.594, -49.433, 81.95, 51.018, -45.38, -40.956] to (141.06, -422.86, -4.17) mm, rotated rx 180 ry 0 rz -179 deg; joints [33.603, -49.407, 81.905, 51.042, -45.375, -40.984]
  MoveL 763 to (141.06, -448.26, -4.17) mm, rotated rx 180 ry 0 rz -179 deg; joints [34.33, -48.494, 80.332, 52.316, -45.448, -42.247]
  MoveL 764 to (90.26, -448.26, -4.18) mm, rotated rx -180 ry 0 rz -179 deg; joints [35.303, -51.243, 85.042, 51.847, -47.298, -40.804]
  MoveL 765 to (90.26, -397.46, -4.17) mm, rotated rx -180 ry 0 rz -179 deg; joints [33.815, -53.016, 88.035, 49.413, -47.123, -38.457]
  MoveL 766 to (141.06, -397.46, -4.17) mm, rotated rx -180 ry 0 rz -179 deg; joints [32.864, -50.289, 83.417, 49.771, -45.297, -39.745]
  MoveL 767 to (141.06, -422.86, -4.17) mm, rotated rx 180 ry 0 rz -179 deg; joints [33.603, -49.407, 81.905, 51.042, -45.375, -40.984]
  MoveC 768 to (140.87, -423.31, -4.17) mm, rotated rx -180 ry 0 rz -179 deg; joints [33.62, -49.401, 81.895, 51.063, -45.383, -41] to (140.42, -423.49, -4.18) mm, rotated rx 180 ry 0 rz -179 deg; joints [33.633, -49.419, 81.926, 51.067, -45.4, -40.996]
  MoveL 769 to (139.79, -423.49, -4.18) mm, rotated rx 180 ry 0 rz -179 deg; joints [33.645, -49.454, 81.987, 51.06, -45.424, -40.977]
  MoveC 770 to (139.34, -423.49, -3.99) mm, rotated rx -180 ry 0 rz -179 deg; joints [33.653, -49.484, 82.024, 51.063, -45.434, -40.975] to (139.15, -423.49, -3.54) mm, rotated rx 180 ry 0 rz -179 deg; joints [33.657, -49.507, 82.029, 51.08, -45.425, -40.997]
  Set speed (500.0 mm/s)
  MoveL 771 to (139.15, -423.49, 5) mm, rotated rx -180 ry 0 rz -179 deg; joints [33.657, -49.736, 81.788, 51.444, -45.13, -41.514]
  MoveL 772 to (139.15, -422.22, 5) mm, rotated rx -180 ry 0 rz -179 deg; joints [33.62, -49.781, 81.865, 51.38, -45.126, -41.451]
  Set speed (25.4 mm/s)
  MoveL 773 to (139.15, -422.22, 1.83) mm, rotated rx -180 ry 0 rz -179 deg; joints [33.62, -49.696, 81.955, 51.244, -45.236, -41.258]
  MoveL 774 to (139.15, -422.22, -7.72) mm, rotated rx -180 ry 0 rz -179 deg; joints [33.62, -49.438, 82.222, 50.842, -45.566, -40.685]
  MoveC 775 to (139.34, -422.22, -8.16) mm, rotated rx -180 ry 0 rz -179 deg; joints [33.617, -49.415, 82.216, 50.825, -45.575, -40.663] to (139.79, -422.22, -8.35) mm, rotated rx -180 ry 0 rz -179 deg; joints [33.608, -49.385, 82.179, 50.822, -45.564, -40.665]
  Set speed (50.8 mm/s)
  MoveL 776 to (140.42, -422.22, -8.35) mm, rotated rx -180 ry 0 rz -179 deg; joints [33.597, -49.35, 82.119, 50.828, -45.541, -40.684]
  MoveC 777 to (140.87, -422.41, -8.35) mm, rotated rx -180 ry 0 rz -179 deg; joints [33.594, -49.319, 82.065, 50.843, -45.525, -40.706] to (141.06, -422.86, -8.35) mm, rotated rx -180 ry 0 rz -179 deg; joints [33.603, -49.293, 82.02, 50.867, -45.519, -40.734]
  MoveL 778 to (141.06, -448.26, -8.35) mm, rotated rx -180 ry 0 rz -179 deg; joints [34.33, -48.383, 80.449, 52.139, -45.588, -41.994]
  MoveL 779 to (90.26, -448.26, -8.35) mm, rotated rx -180 ry 0 rz -179 deg; joints [35.303, -51.125, 85.155, 51.68, -47.442, -40.556]
  MoveL 780 to (90.26, -397.46, -8.35) mm, rotated rx -180 ry 0 rz -179 deg; joints [33.815, -52.894, 88.147, 49.248, -47.276, -38.215]
  MoveL 781 to (141.06, -397.46, -8.35) mm, rotated rx -180 ry 0 rz -179 deg; joints [32.864, -50.173, 83.531, 49.598, -45.446, -39.498]
  MoveL 782 to (141.06, -422.86, -8.35) mm, rotated rx -180 ry 0 rz -179 deg; joints [33.603, -49.293, 82.02, 50.867, -45.519, -40.734]
  MoveC 783 to (140.87, -423.31, -8.35) mm, rotated rx -180 ry 0 rz -179 deg; joints [33.62, -49.287, 82.011, 50.887, -45.527, -40.75] to (140.42, -423.49, -8.35) mm, rotated rx 180 ry 0 rz -179 deg; joints [33.633, -49.306, 82.042, 50.892, -45.544, -40.746]
  MoveL 784 to (139.79, -423.49, -8.35) mm, rotated rx -180 ry 0 rz -179 deg; joints [33.645, -49.34, 82.102, 50.885, -45.568, -40.728]
  MoveC 785 to (139.34, -423.49, -8.16) mm, rotated rx -180 ry 0 rz -179 deg; joints [33.653, -49.37, 82.14, 50.888, -45.578, -40.725] to (139.15, -423.49, -7.72) mm, rotated rx 180 ry 0 rz -179 deg; joints [33.657, -49.393, 82.145, 50.905, -45.57, -40.747]
  Set speed (500.0 mm/s)
  MoveL 786 to (139.15, -423.49, 6) mm, rotated rx -180 ry 0 rz -179 deg; joints [33.657, -49.763, 81.759, 51.487, -45.096, -41.575]
  MoveL 787 to (-92.16, -422.22, 6) mm, rotated rx -180 ry 0 rz -179 deg; joints [38.449, -61.471, 100.951, 51.314, -52.809, -37.048]
  Set speed (25.4 mm/s)
  MoveL 788 to (-92.16, -422.22, -3.54) mm, rotated rx 180 ry 0 rz -179 deg; joints [38.449, -61.152, 101.208, 50.975, -53.17, -36.487]
  MoveC 789 to (-91.98, -422.22, -3.99) mm, rotated rx -180 ry 0 rz -179 deg; joints [38.445, -61.128, 101.206, 50.958, -53.181, -36.463] to (-91.53, -422.22, -4.17) mm, rotated rx 180 ry 0 rz -179 deg; joints [38.435, -61.101, 101.178, 50.948, -53.175, -36.457]
  Set speed (50.8 mm/s)
  MoveL 790 to (-90.89, -422.22, -4.17) mm, rotated rx -180 ry 0 rz -179 deg; joints [38.42, -61.072, 101.132, 50.943, -53.155, -36.464]
  MoveC 791 to (-90.44, -422.41, -4.17) mm, rotated rx -180 ry 0 rz -179 deg; joints [38.415, -61.045, 101.089, 50.947, -53.142, -36.476] to (-90.26, -422.86, -4.17) mm, rotated rx -180 ry 0 rz -179 deg; joints [38.424, -61.02, 101.051, 50.965, -53.139, -36.496]
  MoveL 792 to (-90.26, -448.26, -4.17) mm, rotated rx -180 ry 0 rz -179 deg; joints [39.195, -60.109, 99.613, 52.042, -53.275, -37.471]
  MoveL 793 to (-141.06, -448.26, -4.17) mm, rotated rx -180 ry 0 rz -179 deg; joints [40.429, -62.417, 103.231, 52.505, -54.823, -36.904]
  MoveL 794 to (-141.06, -397.46, -4.17) mm, rotated rx -180 ry 0 rz -179 deg; joints [38.854, -64.251, 106.048, 50.397, -54.509, -35.058]
  MoveL 795 to (-90.26, -397.46, -4.18) mm, rotated rx -180 ry 0 rz -179 deg; joints [37.637, -61.911, 102.445, 49.876, -52.997, -35.532]
  MoveL 796 to (-90.26, -422.86, -4.17) mm, rotated rx -180 ry 0 rz -179 deg; joints [38.424, -61.02, 101.051, 50.965, -53.139, -36.496]
  MoveC 797 to (-90.44, -423.31, -4.17) mm, rotated rx 180 ry 0 rz -179 deg; joints [38.442, -61.013, 101.039, 50.985, -53.147, -36.511] to (-90.89, -423.49, -4.17) mm, rotated rx -180 ry 0 rz -179 deg; joints [38.459, -61.027, 101.061, 50.997, -53.162, -36.513]
  MoveL 798 to (-91.53, -423.49, -4.17) mm, rotated rx -180 ry 0 rz -179 deg; joints [38.474, -61.056, 101.108, 51.002, -53.182, -36.505]
  MoveC 799 to (-91.98, -423.49, -3.99) mm, rotated rx -180 ry 0 rz -179 deg; joints [38.484, -61.083, 101.135, 51.012, -53.188, -36.511] to (-92.16, -423.49, -3.54) mm, rotated rx -180 ry 0 rz -179 deg; joints [38.488, -61.107, 101.137, 51.03, -53.177, -36.535]
  Set speed (500.0 mm/s)
  MoveL 800 to (-92.16, -423.49, 5) mm, rotated rx 180 ry 0 rz -179 deg; joints [38.488, -61.393, 100.907, 51.332, -52.854, -37.038]
  MoveL 801 to (-92.16, -422.22, 5) mm, rotated rx 180 ry 0 rz -179 deg; joints [38.449, -61.438, 100.978, 51.278, -52.846, -36.989]
  Set speed (25.4 mm/s)
  MoveL 802 to (-92.16, -422.22, 1.83) mm, rotated rx -180 ry 0 rz -179 deg; joints [38.449, -61.332, 101.064, 51.165, -52.966, -36.802]
  MoveL 803 to (-92.16, -422.22, -7.72) mm, rotated rx -180 ry 0 rz -179 deg; joints [38.449, -61.011, 101.318, 50.83, -53.328, -36.243]
  MoveC 804 to (-91.98, -422.22, -8.16) mm, rotated rx -180 ry 0 rz -179 deg; joints [38.445, -60.987, 101.316, 50.813, -53.34, -36.219] to (-91.53, -422.22, -8.35) mm, rotated rx -180 ry 0 rz -179 deg; joints [38.435, -60.96, 101.288, 50.802, -53.333, -36.214]
  Set speed (50.8 mm/s)
  MoveL 805 to (-90.89, -422.22, -8.35) mm, rotated rx -180 ry 0 rz -179 deg; joints [38.42, -60.931, 101.242, 50.797, -53.314, -36.221]
  MoveC 806 to (-90.44, -422.41, -8.35) mm, rotated rx -180 ry 0 rz -179 deg; joints [38.415, -60.903, 101.199, 50.801, -53.301, -36.233] to (-90.26, -422.86, -8.35) mm, rotated rx -180 ry 0 rz -179 deg; joints [38.424, -60.879, 101.16, 50.819, -53.298, -36.252]
  MoveL 807 to (-90.26, -448.26, -8.35) mm, rotated rx -180 ry 0 rz -179 deg; joints [39.195, -59.97, 99.722, 51.896, -53.429, -37.227]
  MoveL 808 to (-141.06, -448.26, -8.35) mm, rotated rx -180 ry 0 rz -179 deg; joints [40.429, -62.272, 103.341, 52.363, -54.978, -36.657]
  MoveL 809 to (-141.06, -397.46, -8.35) mm, rotated rx 180 ry 0 rz -179 deg; joints [38.854, -64.101, 106.158, 50.255, -54.675, -34.812]
  MoveL 810 to (-90.26, -397.46, -8.35) mm, rotated rx -180 ry 0 rz -179 deg; joints [37.637, -61.768, 102.555, 49.731, -53.16, -35.29]
  MoveL 811 to (-90.26, -422.86, -8.35) mm, rotated rx -180 ry 0 rz -179 deg; joints [38.424, -60.879, 101.16, 50.819, -53.298, -36.252]
  MoveC 812 to (-90.44, -423.31, -8.35) mm, rotated rx 180 ry 0 rz -179 deg; joints [38.442, -60.871, 101.149, 50.84, -53.306, -36.267] to (-90.89, -423.49, -8.35) mm, rotated rx 180 ry 0 rz -179 deg; joints [38.459, -60.886, 101.171, 50.851, -53.32, -36.269]
  MoveL 813 to (-91.53, -423.49, -8.35) mm, rotated rx -180 ry 0 rz -179 deg; joints [38.474, -60.915, 101.218, 50.856, -53.34, -36.262]
  MoveC 814 to (-91.98, -423.49, -8.16) mm, rotated rx -180 ry 0 rz -179 deg; joints [38.484, -60.942, 101.245, 50.867, -53.347, -36.268] to (-92.16, -423.49, -7.72) mm, rotated rx -180 ry 0 rz -179 deg; joints [38.488, -60.966, 101.247, 50.884, -53.335, -36.292]
  Set speed (500.0 mm/s)
  MoveL 815 to (-92.16, -423.49, 6) mm, rotated rx 180 ry 0 rz -179 deg; joints [38.488, -61.426, 100.88, 51.368, -52.816, -37.097]
  MoveL 816 to (-219.16, -422.22, 6) mm, rotated rx -180 ry 0 rz -179 deg; joints [41.652, -67.203, 109.635, 52.817, -56.531, -36.017]
  Set speed (25.4 mm/s)
  MoveL 817 to (-219.16, -422.22, -3.54) mm, rotated rx 180 ry 0 rz -179 deg; joints [41.652, -66.85, 109.896, 52.497, -56.903, -35.434]
  MoveC 818 to (-218.98, -422.22, -3.99) mm, rotated rx 180 ry 0 rz -179 deg; joints [41.647, -66.825, 109.896, 52.479, -56.915, -35.408] to (-218.53, -422.22, -4.17) mm, rotated rx -180 ry 0 rz -179 deg; joints [41.635, -66.799, 109.872, 52.466, -56.91, -35.399]
  Set speed (50.8 mm/s)
  MoveL 819 to (-217.89, -422.22, -4.17) mm, rotated rx -180 ry 0 rz -179 deg; joints [41.618, -66.771, 109.831, 52.456, -56.892, -35.403]
  MoveC 820 to (-217.44, -422.41, -4.18) mm, rotated rx 180 ry 0 rz -179 deg; joints [41.611, -66.745, 109.792, 52.457, -56.88, -35.411] to (-217.26, -422.86, -4.18) mm, rotated rx -180 ry 0 rz -179 deg; joints [41.62, -66.72, 109.755, 52.472, -56.878, -35.427]
  MoveL 821 to (-217.26, -448.26, -4.18) mm, rotated rx 180 ry 0 rz -179 deg; joints [42.409, -65.763, 108.331, 53.477, -57.058, -36.288]
  MoveL 822 to (-268.06, -448.26, -4.18) mm, rotated rx -180 ry 0 rz -179 deg; joints [43.821, -67.925, 111.527, 54.298, -58.502, -36.019]
  MoveL 823 to (-268.06, -397.46, -4.17) mm, rotated rx 180 ry 0 rz -179 deg; joints [42.215, -69.874, 114.341, 52.327, -58.092, -34.393]
  MoveL 824 to (-217.26, -397.46, -4.18) mm, rotated rx 180 ry 0 rz -179 deg; joints [40.813, -67.66, 111.14, 51.452, -56.689, -34.575]
  MoveL 825 to (-217.26, -422.86, -4.18) mm, rotated rx -180 ry 0 rz -179 deg; joints [41.62, -66.72, 109.755, 52.472, -56.878, -35.427]
  MoveC 826 to (-217.44, -423.31, -4.18) mm, rotated rx 180 ry 0 rz -179 deg; joints [41.639, -66.711, 109.742, 52.493, -56.887, -35.442] to (-217.89, -423.49, -4.18) mm, rotated rx -180 ry 0 rz -179 deg; joints [41.657, -66.724, 109.761, 52.507, -56.901, -35.445]
  MoveL 827 to (-218.53, -423.49, -4.18) mm, rotated rx 180 ry 0 rz -179 deg; joints [41.675, -66.752, 109.802, 52.517, -56.919, -35.442]
  MoveC 828 to (-218.98, -423.49, -3.99) mm, rotated rx -180 ry 0 rz -179 deg; joints [41.687, -66.778, 109.826, 52.53, -56.924, -35.451] to (-219.16, -423.49, -3.54) mm, rotated rx -180 ry 0 rz -179 deg; joints [41.692, -66.803, 109.826, 52.548, -56.912, -35.477]
  Set speed (500.0 mm/s)
  MoveL 829 to (-219.16, -423.49, 5) mm, rotated rx -180 ry 0 rz -179 deg; joints [41.692, -67.119, 109.593, 52.834, -56.58, -35.999]
  MoveL 830 to (-219.16, -422.22, 5) mm, rotated rx 180 ry 0 rz -179 deg; joints [41.652, -67.166, 109.663, 52.783, -56.57, -35.956]
  Set speed (25.4 mm/s)
  MoveL 831 to (-219.16, -422.22, 1.82) mm, rotated rx 180 ry 0 rz -179 deg; joints [41.652, -67.049, 109.75, 52.676, -56.693, -35.761]
  MoveL 832 to (-219.16, -422.22, -7.71) mm, rotated rx 180 ry 0 rz -179 deg; joints [41.652, -66.694, 110.008, 52.359, -57.066, -35.181]
  MoveC 833 to (-218.98, -422.22, -8.16) mm, rotated rx -180 ry 0 rz -179 deg; joints [41.647, -66.669, 110.008, 52.341, -57.079, -35.155] to (-218.53, -422.22, -8.35) mm, rotated rx -180 ry 0 rz -179 deg; joints [41.635, -66.643, 109.984, 52.328, -57.073, -35.146]
  Set speed (50.8 mm/s)
  MoveL 834 to (-217.89, -422.22, -8.35) mm, rotated rx -180 ry 0 rz -179 deg; joints [41.618, -66.615, 109.943, 52.318, -57.055, -35.15]
  MoveC 835 to (-217.44, -422.41, -8.35) mm, rotated rx 180 ry 0 rz -179 deg; joints [41.611, -66.589, 109.903, 52.319, -57.044, -35.158] to (-217.26, -422.86, -8.35) mm, rotated rx 180 ry 0 rz -179 deg; joints [41.62, -66.564, 109.867, 52.334, -57.042, -35.174]
  MoveL 836 to (-217.26, -448.26, -8.35) mm, rotated rx -180 ry 0 rz -179 deg; joints [42.409, -65.61, 108.442, 53.34, -57.216, -36.036]
  MoveL 837 to (-268.06, -448.26, -8.35) mm, rotated rx 180 ry 0 rz -179 deg; joints [43.821, -67.765, 111.639, 54.163, -58.661, -35.761]
  MoveL 838 to (-268.06, -397.46, -8.35) mm, rotated rx 180 ry 0 rz -179 deg; joints [42.215, -69.71, 114.454, 52.191, -58.262, -34.134]
  MoveL 839 to (-217.26, -397.46, -8.35) mm, rotated rx -180 ry 0 rz -179 deg; joints [40.813, -67.502, 111.252, 51.313, -56.858, -34.323]
  MoveL 840 to (-217.26, -422.86, -8.35) mm, rotated rx -180 ry 0 rz -179 deg; joints [41.62, -66.564, 109.867, 52.334, -57.042, -35.174]
  MoveC 841 to (-217.44, -423.31, -8.35) mm, rotated rx 180 ry 0 rz -179 deg; joints [41.639, -66.555, 109.854, 52.355, -57.05, -35.189] to (-217.89, -423.49, -8.35) mm, rotated rx -180 ry 0 rz -179 deg; joints [41.657, -66.568, 109.872, 52.369, -57.064, -35.192]
  MoveL 842 to (-218.53, -423.49, -8.35) mm, rotated rx -180 ry 0 rz -179 deg; joints [41.675, -66.595, 109.913, 52.379, -57.082, -35.189]
  MoveC 843 to (-218.98, -423.49, -8.16) mm, rotated rx 180 ry 0 rz -179 deg; joints [41.687, -66.622, 109.937, 52.392, -57.088, -35.198] to (-219.16, -423.49, -7.72) mm, rotated rx 180 ry 0 rz -179 deg; joints [41.692, -66.647, 109.937, 52.41, -57.075, -35.224]
  Set speed (500.0 mm/s)
  MoveL 844 to (-219.16, -423.49, 6) mm, rotated rx 180 ry 0 rz -179 deg; joints [41.692, -67.155, 109.565, 52.868, -56.541, -36.06]
  MoveL 845 to (-346.16, -422.22, 6) mm, rotated rx 180 ry 0 rz -179 deg; joints [45.333, -72.617, 117.327, 55.186, -60.026, -35.695]
  Set speed (25.4 mm/s)
  MoveL 846 to (-346.16, -422.22, -3.54) mm, rotated rx -180 ry 0 rz -179 deg; joints [45.333, -72.231, 117.596, 54.878, -60.402, -35.076]
  MoveC 847 to (-345.98, -422.22, -3.99) mm, rotated rx 180 ry 0 rz -179 deg; joints [45.327, -72.205, 117.598, 54.86, -60.415, -35.047] to (-345.53, -422.22, -4.17) mm, rotated rx -180 ry 0 rz -179 deg; joints [45.313, -72.178, 117.577, 54.844, -60.41, -35.035]
  Set speed (50.8 mm/s)
  MoveL 848 to (-344.89, -422.22, -4.18) mm, rotated rx 180 ry 0 rz -179 deg; joints [45.293, -72.152, 117.541, 54.83, -60.393, -35.036]
  MoveC 849 to (-344.44, -422.41, -4.18) mm, rotated rx -180 ry 0 rz -179 deg; joints [45.285, -72.126, 117.505, 54.827, -60.383, -35.041] to (-344.26, -422.86, -4.17) mm, rotated rx -180 ry 0 rz -179 deg; joints [45.294, -72.101, 117.47, 54.84, -60.382, -35.055]
  MoveL 850 to (-344.26, -448.26, -4.18) mm, rotated rx -180 ry 0 rz -179 deg; joints [46.09, -71.072, 116.036, 55.774, -60.613, -35.805]
  MoveL 851 to (-395.06, -448.26, -4.17) mm, rotated rx -180 ry 0 rz -179 deg; joints [47.709, -73.11, 118.858, 56.914, -61.994, -35.78]
  MoveL 852 to (-395.06, -397.46, -4.17) mm, rotated rx -180 ry 0 rz -179 deg; joints [46.095, -75.229, 121.706, 55.089, -61.475, -34.382]
  MoveL 853 to (-344.26, -397.46, -4.18) mm, rotated rx 180 ry 0 rz -179 deg; joints [44.475, -73.117, 118.867, 53.888, -60.138, -34.313]
  MoveL 854 to (-344.26, -422.86, -4.17) mm, rotated rx -180 ry 0 rz -179 deg; joints [45.294, -72.101, 117.47, 54.84, -60.382, -35.055]
  MoveC 855 to (-344.44, -423.31, -4.18) mm, rotated rx 180 ry 0 rz -179 deg; joints [45.314, -72.09, 117.455, 54.86, -60.391, -35.068] to (-344.89, -423.49, -4.18) mm, rotated rx -180 ry 0 rz -179 deg; joints [45.334, -72.101, 117.47, 54.877, -60.405, -35.073]
  MoveL 856 to (-345.53, -423.49, -4.18) mm, rotated rx -180 ry 0 rz -179 deg; joints [45.353, -72.127, 117.507, 54.891, -60.422, -35.073]
  MoveC 857 to (-345.98, -423.49, -3.99) mm, rotated rx 180 ry 0 rz -179 deg; joints [45.367, -72.153, 117.527, 54.907, -60.427, -35.084] to (-346.16, -423.49, -3.54) mm, rotated rx 180 ry 0 rz -179 deg; joints [45.373, -72.179, 117.525, 54.925, -60.414, -35.113]
  Set speed (500.0 mm/s)
  MoveL 858 to (-346.16, -423.49, 5) mm, rotated rx 180 ry 0 rz -179 deg; joints [45.373, -72.526, 117.285, 55.2, -60.078, -35.667]
  MoveL 859 to (-346.16, -422.22, 5) mm, rotated rx -180 ry 0 rz -179 deg; joints [45.333, -72.577, 117.355, 55.153, -60.066, -35.63]
  Set speed (25.4 mm/s)
  MoveL 860 to (-346.16, -422.22, 1.82) mm, rotated rx -180 ry 0 rz -179 deg; joints [45.333, -72.449, 117.445, 55.05, -60.19, -35.424]
  MoveL 861 to (-346.16, -422.22, -7.72) mm, rotated rx -180 ry 0 rz -179 deg; joints [45.333, -72.059, 117.711, 54.745, -60.568, -34.807]
  MoveC 862 to (-345.98, -422.22, -8.16) mm, rotated rx -180 ry 0 rz -179 deg; joints [45.327, -72.033, 117.713, 54.727, -60.58, -34.778] to (-345.53, -422.22, -8.35) mm, rotated rx 180 ry 0 rz -179 deg; joints [45.313, -72.007, 117.693, 54.711, -60.576, -34.766]
  Set speed (50.8 mm/s)
  MoveL 863 to (-344.89, -422.22, -8.35) mm, rotated rx -180 ry 0 rz -179 deg; joints [45.293, -71.981, 117.656, 54.697, -60.559, -34.767]
  MoveC 864 to (-344.44, -422.41, -8.35) mm, rotated rx -180 ry 0 rz -179 deg; joints [45.285, -71.955, 117.62, 54.694, -60.548, -34.772] to (-344.26, -422.86, -8.35) mm, rotated rx -180 ry 0 rz -179 deg; joints [45.294, -71.929, 117.585, 54.707, -60.547, -34.786]
  MoveL 865 to (-344.26, -448.26, -8.35) mm, rotated rx 180 ry 0 rz -179 deg; joints [46.09, -70.904, 116.15, 55.643, -60.772, -35.537]
  MoveL 866 to (-395.06, -448.26, -8.35) mm, rotated rx -180 ry 0 rz -179 deg; joints [47.709, -72.936, 118.974, 56.785, -62.153, -35.505]
  MoveL 867 to (-395.06, -397.46, -8.35) mm, rotated rx 180 ry 0 rz -179 deg; joints [46.095, -75.048, 121.825, 54.956, -61.646, -34.104]
  MoveL 868 to (-344.26, -397.46, -8.35) mm, rotated rx -180 ry 0 rz -179 deg; joints [44.475, -72.943, 118.983, 53.754, -60.31, -34.043]
  MoveL 869 to (-344.26, -422.86, -8.35) mm, rotated rx -180 ry 0 rz -179 deg; joints [45.294, -71.929, 117.585, 54.707, -60.547, -34.786]
  MoveC 870 to (-344.44, -423.31, -8.35) mm, rotated rx -180 ry 0 rz -179 deg; joints [45.314, -71.919, 117.57, 54.728, -60.556, -34.799] to (-344.89, -423.49, -8.35) mm, rotated rx -180 ry 0 rz -179 deg; joints [45.334, -71.93, 117.586, 54.745, -60.57, -34.804]
  MoveL 871 to (-345.53, -423.49, -8.35) mm, rotated rx -180 ry 0 rz -179 deg; joints [45.353, -71.956, 117.622, 54.758, -60.587, -34.803]
  MoveC 872 to (-345.98, -423.49, -8.16) mm, rotated rx -180 ry 0 rz -179 deg; joints [45.367, -71.982, 117.642, 54.774, -60.592, -34.815] to (-346.16, -423.49, -7.72) mm, rotated rx -180 ry 0 rz -179 deg; joints [45.373, -72.008, 117.641, 54.792, -60.579, -34.844]
  Set speed (500.0 mm/s)
  MoveL 873 to (-346.16, -423.49, 6) mm, rotated rx 180 ry 0 rz -179 deg; joints [45.373, -72.566, 117.256, 55.233, -60.039, -35.732]
  MoveL 874 to (-346.16, -235.88, 6) mm, rotated rx 180 ry 0 rz -179 deg; joints [38.77, -79.853, 126.727, 47.737, -57.792, -30.392]
  Set speed (25.4 mm/s)
  MoveL 875 to (-346.16, -235.89, -3.54) mm, rotated rx 180 ry 0 rz -179 deg; joints [38.77, -79.417, 127.015, 47.404, -58.281, -29.763]
  MoveC 876 to (-345.98, -235.89, -3.99) mm, rotated rx 180 ry 0 rz -179 deg; joints [38.764, -79.388, 127.017, 47.384, -58.3, -29.732] to (-345.53, -235.88, -4.17) mm, rotated rx 180 ry 0 rz -179 deg; joints [38.75, -79.358, 126.996, 47.366, -58.299, -29.717]
  Set speed (50.8 mm/s)
  MoveL 877 to (-344.89, -235.89, -4.18) mm, rotated rx -180 ry 0 rz -179 deg; joints [38.731, -79.328, 126.959, 47.35, -58.285, -29.713]
  MoveC 878 to (-344.44, -236.07, -4.17) mm, rotated rx -180 ry 0 rz -179 deg; joints [38.725, -79.3, 126.924, 47.346, -58.277, -29.715] to (-344.26, -236.52, -4.18) mm, rotated rx -180 ry 0 rz -179 deg; joints [38.737, -79.274, 126.893, 47.361, -58.279, -29.727]
  MoveL 879 to (-344.26, -261.92, -4.18) mm, rotated rx -180 ry 0 rz -179 deg; joints [39.709, -78.337, 125.721, 48.455, -58.609, -30.447]
  MoveL 880 to (-395.06, -261.92, -4.18) mm, rotated rx 180 ry 0 rz -179 deg; joints [41.3, -80.688, 128.625, 49.8, -59.78, -30.778]
  MoveL 881 to (-395.06, -211.12, -4.18) mm, rotated rx -180 ry 0 rz -179 deg; joints [39.304, -82.655, 130.961, 47.63, -59.023, -29.434]
  MoveL 882 to (-344.26, -211.12, -4.17) mm, rotated rx -180 ry 0 rz -179 deg; joints [37.738, -80.198, 128.029, 46.24, -57.934, -29.003]
  MoveL 883 to (-344.26, -236.52, -4.18) mm, rotated rx -180 ry 0 rz -179 deg; joints [38.737, -79.274, 126.893, 47.361, -58.279, -29.727]
  MoveC 884 to (-344.44, -236.97, -4.17) mm, rotated rx -180 ry 0 rz -179 deg; joints [38.76, -79.267, 126.884, 47.385, -58.289, -29.741] to (-344.89, -237.16, -4.18) mm, rotated rx -180 ry 0 rz -179 deg; joints [38.781, -79.281, 126.901, 47.405, -58.302, -29.749]
  MoveL 885 to (-345.53, -237.15, -4.18) mm, rotated rx 180 ry 0 rz -179 deg; joints [38.8, -79.311, 126.939, 47.421, -58.316, -29.753]
  MoveC 886 to (-345.98, -237.16, -3.99) mm, rotated rx -180 ry 0 rz -179 deg; joints [38.813, -79.341, 126.959, 47.439, -58.317, -29.768] to (-346.16, -237.15, -3.54) mm, rotated rx 180 ry 0 rz -179 deg; joints [38.819, -79.371, 126.957, 47.459, -58.298, -29.799]
  Set speed (500.0 mm/s)
  MoveL 887 to (-346.16, -237.15, 5) mm, rotated rx -180 ry 0 rz -179 deg; joints [38.819, -79.761, 126.7, 47.757, -57.861, -30.362]
  MoveL 888 to (-346.16, -235.89, 5) mm, rotated rx 180 ry 0 rz -179 deg; joints [38.77, -79.808, 126.757, 47.702, -57.843, -30.326]
  Set speed (25.4 mm/s)
  MoveL 889 to (-346.16, -235.89, 1.82) mm, rotated rx 180 ry 0 rz -179 deg; joints [38.77, -79.663, 126.854, 47.591, -58.006, -30.116]
  MoveL 890 to (-346.16, -235.88, -7.72) mm, rotated rx 180 ry 0 rz -179 deg; joints [38.77, -79.224, 127.138, 47.261, -58.495, -29.489]
  MoveC 891 to (-345.98, -235.88, -8.16) mm, rotated rx 180 ry 0 rz -179 deg; joints [38.764, -79.194, 127.141, 47.241, -58.514, -29.458] to (-345.53, -235.88, -8.35) mm, rotated rx -180 ry 0 rz -179 deg; joints [38.75, -79.164, 127.12, 47.223, -58.514, -29.444]
  Set speed (50.8 mm/s)
  MoveL 892 to (-344.89, -235.89, -8.35) mm, rotated rx -180 ry 0 rz -179 deg; joints [38.731, -79.134, 127.082, 47.206, -58.5, -29.44]
  MoveC 893 to (-344.44, -236.07, -8.35) mm, rotated rx -180 ry 0 rz -179 deg; joints [38.725, -79.106, 127.048, 47.203, -58.492, -29.442] to (-344.26, -236.52, -8.35) mm, rotated rx -180 ry 0 rz -179 deg; joints [38.737, -79.081, 127.016, 47.218, -58.493, -29.454]
  MoveL 894 to (-344.26, -261.92, -8.35) mm, rotated rx 180 ry 0 rz -179 deg; joints [39.709, -78.146, 125.843, 48.313, -58.817, -30.174]
  MoveL 895 to (-395.06, -261.92, -8.35) mm, rotated rx 180 ry 0 rz -179 deg; joints [41.3, -80.491, 128.75, 49.657, -59.989, -30.493]
  MoveL 896 to (-395.06, -211.12, -8.35) mm, rotated rx -180 ry 0 rz -179 deg; joints [39.304, -82.451, 131.089, 47.483, -59.247, -29.148]
  MoveL 897 to (-344.26, -211.12, -8.35) mm, rotated rx -180 ry 0 rz -179 deg; joints [37.738, -80.002, 128.154, 46.096, -58.157, -28.73]
  MoveL 898 to (-344.26, -236.52, -8.35) mm, rotated rx -180 ry 0 rz -179 deg; joints [38.737, -79.081, 127.016, 47.218, -58.493, -29.454]
  MoveC 899 to (-344.44, -236.97, -8.35) mm, rotated rx -180 ry 0 rz -179 deg; joints [38.76, -79.074, 127.007, 47.242, -58.503, -29.468] to (-344.89, -237.16, -8.35) mm, rotated rx 180 ry 0 rz -179 deg; joints [38.781, -79.088, 127.025, 47.262, -58.516, -29.476]
  MoveL 900 to (-345.53, -237.15, -8.35) mm, rotated rx -180 ry 0 rz -179 deg; joints [38.8, -79.118, 127.062, 47.278, -58.53, -29.48]
  MoveC 901 to (-345.98, -237.16, -8.16) mm, rotated rx -180 ry 0 rz -179 deg; joints [38.813, -79.148, 127.083, 47.296, -58.531, -29.494] to (-346.16, -237.15, -7.72) mm, rotated rx 180 ry 0 rz -179 deg; joints [38.819, -79.177, 127.081, 47.316, -58.512, -29.525]
  Set speed (500.0 mm/s)
  MoveL 902 to (-346.16, -237.16, 6) mm, rotated rx -180 ry 0 rz -179 deg; joints [38.819, -79.806, 126.669, 47.793, -57.81, -30.428]
  MoveL 903 to (-219.16, -235.89, 6) mm, rotated rx -180 ry 0 rz -179 deg; joints [35.255, -73.769, 118.893, 44.928, -54.819, -29.887]
  Set speed (25.4 mm/s)
  MoveL 904 to (-219.16, -235.89, -3.54) mm, rotated rx 180 ry 0 rz -179 deg; joints [35.255, -73.375, 119.164, 44.601, -55.291, -29.315]
  MoveC 905 to (-218.98, -235.89, -3.99) mm, rotated rx -180 ry 0 rz -179 deg; joints [35.25, -73.347, 119.165, 44.582, -55.309, -29.288] to (-218.53, -235.88, -4.17) mm, rotated rx -180 ry 0 rz -179 deg; joints [35.239, -73.318, 119.141, 44.567, -55.307, -29.277]
  Set speed (50.8 mm/s)
  MoveL 906 to (-217.89, -235.88, -4.18) mm, rotated rx 180 ry 0 rz -179 deg; joints [35.223, -73.287, 119.099, 44.556, -55.291, -29.277]
  MoveC 907 to (-217.44, -236.07, -4.17) mm, rotated rx -180 ry 0 rz -179 deg; joints [35.218, -73.26, 119.062, 44.556, -55.282, -29.282] to (-217.26, -236.52, -4.17) mm, rotated rx 180 ry 0 rz -179 deg; joints [35.23, -73.236, 119.03, 44.573, -55.282, -29.297]
  MoveL 908 to (-217.26, -261.92, -4.18) mm, rotated rx -180 ry 0 rz -179 deg; joints [36.167, -72.401, 117.885, 45.712, -55.527, -30.125]
  MoveL 909 to (-268.06, -261.92, -4.17) mm, rotated rx -180 ry 0 rz -179 deg; joints [37.514, -74.787, 121.12, 46.704, -56.792, -30.168]
  MoveL 910 to (-268.06, -211.12, -4.18) mm, rotated rx -180 ry 0 rz -179 deg; joints [35.588, -76.515, 123.391, 44.434, -56.228, -28.591]
  MoveL 911 to (-217.26, -211.12, -4.18) mm, rotated rx 180 ry 0 rz -179 deg; joints [34.273, -74.054, 120.138, 43.411, -55.028, -28.468]
  MoveL 912 to (-217.26, -236.52, -4.17) mm, rotated rx 180 ry 0 rz -179 deg; joints [35.23, -73.236, 119.03, 44.573, -55.282, -29.297]
  MoveC 913 to (-217.44, -236.97, -4.18) mm, rotated rx 180 ry 0 rz -179 deg; joints [35.252, -73.231, 119.022, 44.596, -55.291, -29.312] to (-217.89, -237.15, -4.18) mm, rotated rx 180 ry 0 rz -179 deg; joints [35.27, -73.246, 119.043, 44.613, -55.304, -29.318]
  MoveL 914 to (-218.53, -237.15, -4.18) mm, rotated rx 180 ry 0 rz -179 deg; joints [35.286, -73.276, 119.084, 44.625, -55.32, -29.318]
  MoveC 915 to (-218.98, -237.15, -3.99) mm, rotated rx -180 ry 0 rz -179 deg; joints [35.298, -73.306, 119.108, 44.639, -55.322, -29.33] to (-219.16, -237.16, -3.54) mm, rotated rx 180 ry 0 rz -179 deg; joints [35.302, -73.333, 119.108, 44.658, -55.304, -29.357]
  Set speed (500.0 mm/s)
  MoveL 916 to (-219.16, -237.16, 5) mm, rotated rx -180 ry 0 rz -179 deg; joints [35.302, -73.686, 118.865, 44.951, -54.881, -29.868]
  MoveL 917 to (-219.16, -235.89, 5) mm, rotated rx 180 ry 0 rz -179 deg; joints [35.255, -73.728, 118.921, 44.894, -54.868, -29.827]
  Set speed (25.4 mm/s)
  MoveL 918 to (-219.16, -235.89, 1.83) mm, rotated rx 180 ry 0 rz -179 deg; joints [35.255, -73.597, 119.012, 44.784, -55.025, -29.636]
  MoveL 919 to (-219.16, -235.89, -7.72) mm, rotated rx 180 ry 0 rz -179 deg; joints [35.255, -73.2, 119.281, 44.46, -55.499, -29.067]
  MoveC 920 to (-218.98, -235.89, -8.16) mm, rotated rx -180 ry 0 rz -179 deg; joints [35.25, -73.172, 119.281, 44.441, -55.517, -29.04] to (-218.53, -235.89, -8.35) mm, rotated rx 180 ry 0 rz -179 deg; joints [35.239, -73.143, 119.257, 44.427, -55.515, -29.029]
  Set speed (50.8 mm/s)
  MoveL 921 to (-217.89, -235.89, -8.35) mm, rotated rx -180 ry 0 rz -179 deg; joints [35.223, -73.113, 119.216, 44.415, -55.499, -29.029]
  MoveC 922 to (-217.44, -236.07, -8.35) mm, rotated rx 180 ry 0 rz -179 deg; joints [35.218, -73.085, 119.178, 44.415, -55.49, -29.035] to (-217.26, -236.52, -8.35) mm, rotated rx -180 ry 0 rz -179 deg; joints [35.23, -73.062, 119.146, 44.432, -55.489, -29.049]
  MoveL 923 to (-217.26, -261.92, -8.35) mm, rotated rx 180 ry 0 rz -179 deg; joints [36.167, -72.229, 118, 45.571, -55.729, -29.875]
  MoveL 924 to (-268.06, -261.92, -8.35) mm, rotated rx 180 ry 0 rz -179 deg; joints [37.514, -74.608, 121.238, 46.563, -56.996, -29.91]
  MoveL 925 to (-268.06, -211.12, -8.35) mm, rotated rx -180 ry 0 rz -179 deg; joints [35.588, -76.33, 123.511, 44.292, -56.445, -28.336]
  MoveL 926 to (-217.26, -211.12, -8.35) mm, rotated rx 180 ry 0 rz -179 deg; joints [34.273, -73.877, 120.255, 43.27, -55.242, -28.222]
  MoveL 927 to (-217.26, -236.52, -8.35) mm, rotated rx 180 ry 0 rz -179 deg; joints [35.23, -73.062, 119.146, 44.432, -55.489, -29.049]
  MoveC 928 to (-217.44, -236.97, -8.35) mm, rotated rx 180 ry 0 rz -179 deg; joints [35.252, -73.056, 119.138, 44.456, -55.498, -29.064] to (-217.89, -237.16, -8.35) mm, rotated rx -180 ry 0 rz -179 deg; joints [35.27, -73.071, 119.159, 44.472, -55.511, -29.07]
  MoveL 929 to (-218.53, -237.16, -8.35) mm, rotated rx -180 ry 0 rz -179 deg; joints [35.286, -73.102, 119.201, 44.484, -55.527, -29.07]
  MoveC 930 to (-218.98, -237.15, -8.16) mm, rotated rx 180 ry 0 rz -179 deg; joints [35.298, -73.131, 119.225, 44.499, -55.529, -29.082] to (-219.16, -237.16, -7.72) mm, rotated rx 180 ry 0 rz -179 deg; joints [35.302, -73.159, 119.224, 44.517, -55.511, -29.108]
  Set speed (500.0 mm/s)
  MoveL 931 to (-219.16, -237.15, 6) mm, rotated rx -180 ry 0 rz -179 deg; joints [35.302, -73.727, 118.836, 44.986, -54.832, -29.929]
  MoveL 932 to (-92.16, -235.89, 6) mm, rotated rx -180 ry 0 rz -179 deg; joints [32.277, -67.587, 110.199, 43.012, -51.52, -30.135]
  Set speed (25.4 mm/s)
  MoveL 933 to (-92.16, -235.88, -3.54) mm, rotated rx 180 ry 0 rz -179 deg; joints [32.277, -67.233, 110.46, 42.682, -51.971, -29.602]
  MoveC 934 to (-91.98, -235.88, -3.99) mm, rotated rx -180 ry 0 rz -179 deg; joints [32.273, -67.207, 110.458, 42.664, -51.988, -29.578] to (-91.53, -235.88, -4.17) mm, rotated rx -180 ry 0 rz -179 deg; joints [32.263, -67.178, 110.431, 42.653, -51.984, -29.57]
  Set speed (50.8 mm/s)
  MoveL 935 to (-90.89, -235.89, -4.17) mm, rotated rx -180 ry 0 rz -179 deg; joints [32.249, -67.146, 110.385, 42.645, -51.966, -29.573]
  MoveC 936 to (-90.44, -236.07, -4.18) mm, rotated rx 180 ry 0 rz -179 deg; joints [32.246, -67.119, 110.345, 42.649, -51.955, -29.582] to (-90.26, -236.52, -4.17) mm, rotated rx 180 ry 0 rz -179 deg; joints [32.258, -67.096, 110.311, 42.668, -51.953, -29.6]
  MoveL 937 to (-90.26, -261.92, -4.18) mm, rotated rx 180 ry 0 rz -179 deg; joints [33.152, -66.331, 109.177, 43.847, -52.133, -30.524]
  MoveL 938 to (-141.06, -261.92, -4.17) mm, rotated rx -180 ry 0 rz -179 deg; joints [34.301, -68.781, 112.771, 44.486, -53.535, -30.275]
  MoveL 939 to (-141.06, -211.12, -4.17) mm, rotated rx -180 ry 0 rz -179 deg; joints [32.46, -70.342, 115.005, 42.141, -53.121, -28.504]
  MoveL 940 to (-90.26, -211.12, -4.18) mm, rotated rx 180 ry 0 rz -179 deg; joints [31.346, -67.842, 111.406, 41.472, -51.769, -28.677]
  MoveL 941 to (-90.26, -236.52, -4.17) mm, rotated rx 180 ry 0 rz -179 deg; joints [32.258, -67.096, 110.311, 42.668, -51.953, -29.6]
  MoveC 942 to (-90.44, -236.97, -4.17) mm, rotated rx -180 ry 0 rz -179 deg; joints [32.278, -67.092, 110.305, 42.691, -51.962, -29.615] to (-90.89, -237.15, -4.17) mm, rotated rx -180 ry 0 rz -179 deg; joints [32.294, -67.109, 110.33, 42.705, -51.976, -29.619]
  MoveL 943 to (-91.53, -237.16, -4.17) mm, rotated rx -180 ry 0 rz -179 deg; joints [32.308, -67.14, 110.375, 42.712, -51.993, -29.616]
  MoveC 944 to (-91.98, -237.16, -3.99) mm, rotated rx 180 ry 0 rz -179 deg; joints [32.318, -67.169, 110.403, 42.724, -51.997, -29.624] to (-92.16, -237.15, -3.54) mm, rotated rx -180 ry 0 rz -179 deg; joints [32.322, -67.195, 110.404, 42.741, -51.981, -29.648]
  Set speed (500.0 mm/s)
  MoveL 945 to (-92.16, -237.15, 5) mm, rotated rx 180 ry 0 rz -179 deg; joints [32.322, -67.513, 110.171, 43.037, -51.577, -30.125]
  MoveL 946 to (-92.16, -235.89, 5) mm, rotated rx 180 ry 0 rz -179 deg; joints [32.277, -67.551, 110.226, 42.977, -51.567, -30.079]
  Set speed (25.4 mm/s)
  MoveL 947 to (-92.16, -235.89, 1.82) mm, rotated rx 180 ry 0 rz -179 deg; joints [32.277, -67.433, 110.314, 42.867, -51.717, -29.901]
  MoveL 948 to (-92.16, -235.89, -7.72) mm, rotated rx -180 ry 0 rz -179 deg; joints [32.277, -67.075, 110.572, 42.54, -52.17, -29.371]
  MoveC 949 to (-91.98, -235.89, -8.16) mm, rotated rx -180 ry 0 rz -179 deg; joints [32.273, -67.049, 110.57, 42.522, -52.186, -29.347] to (-91.53, -235.88, -8.35) mm, rotated rx -180 ry 0 rz -179 deg; joints [32.263, -67.02, 110.543, 42.511, -52.182, -29.339]
  Set speed (50.8 mm/s)
  MoveL 950 to (-90.89, -235.89, -8.35) mm, rotated rx 180 ry 0 rz -179 deg; joints [32.249, -66.989, 110.497, 42.504, -52.164, -29.342]
  MoveC 951 to (-90.44, -236.07, -8.35) mm, rotated rx 180 ry 0 rz -179 deg; joints [32.246, -66.962, 110.456, 42.507, -52.153, -29.352] to (-90.26, -236.52, -8.35) mm, rotated rx -180 ry 0 rz -179 deg; joints [32.258, -66.939, 110.423, 42.526, -52.151, -29.369]
  MoveL 952 to (-90.26, -261.92, -8.35) mm, rotated rx 180 ry 0 rz -179 deg; joints [33.152, -66.176, 109.289, 43.704, -52.325, -30.29]
  MoveL 953 to (-141.06, -261.92, -8.35) mm, rotated rx -180 ry 0 rz -179 deg; joints [34.301, -68.619, 112.884, 44.345, -53.731, -30.036]
  MoveL 954 to (-141.06, -211.12, -8.35) mm, rotated rx -180 ry 0 rz -179 deg; joints [32.46, -70.175, 115.119, 42.001, -53.329, -28.27]
  MoveL 955 to (-90.26, -211.12, -8.35) mm, rotated rx 180 ry 0 rz -179 deg; joints [31.346, -67.683, 111.518, 41.331, -51.972, -28.449]
  MoveL 956 to (-90.26, -236.52, -8.35) mm, rotated rx -180 ry 0 rz -179 deg; joints [32.258, -66.939, 110.423, 42.526, -52.151, -29.369]
  MoveC 957 to (-90.44, -236.97, -8.35) mm, rotated rx 180 ry 0 rz -179 deg; joints [32.278, -66.935, 110.417, 42.549, -52.16, -29.384] to (-90.89, -237.16, -8.35) mm, rotated rx 180 ry 0 rz -179 deg; joints [32.294, -66.951, 110.441, 42.563, -52.173, -29.388]
  MoveL 958 to (-91.53, -237.16, -8.35) mm, rotated rx -180 ry 0 rz -179 deg; joints [32.308, -66.983, 110.487, 42.57, -52.191, -29.385]
  MoveC 959 to (-91.98, -237.16, -8.16) mm, rotated rx 180 ry 0 rz -179 deg; joints [32.318, -67.011, 110.515, 42.582, -52.195, -29.393] to (-92.16, -237.16, -7.72) mm, rotated rx -180 ry 0 rz -179 deg; joints [32.322, -67.038, 110.516, 42.599, -52.179, -29.417]
  Set speed (500.0 mm/s)
  MoveL 960 to (-92.16, -237.15, 6) mm, rotated rx 180 ry 0 rz -179 deg; joints [32.322, -67.549, 110.143, 43.072, -51.53, -30.181]
  MoveL 961 to (-92.16, -54.85, 6) mm, rotated rx -180 ry 0 rz -179 deg; joints [25.394, -72.481, 117.14, 34.033, -50.015, -23.46]
  Set speed (25.4 mm/s)
  MoveL 962 to (-92.16, -54.85, -3.54) mm, rotated rx -180 ry 0 rz -179 deg; joints [25.394, -72.095, 117.409, 33.73, -50.559, -22.985]
  MoveC 963 to (-91.98, -54.85, -3.99) mm, rotated rx 180 ry 0 rz -179 deg; joints [25.39, -72.067, 117.408, 33.714, -50.58, -22.963] to (-91.53, -54.85, -4.17) mm, rotated rx 180 ry 0 rz -179 deg; joints [25.382, -72.036, 117.38, 33.702, -50.58, -22.954]
  Set speed (50.8 mm/s)
  MoveL 964 to (-90.89, -54.85, -4.17) mm, rotated rx -180 ry 0 rz -179 deg; joints [25.37, -72.003, 117.334, 33.694, -50.565, -22.955]
  MoveC 965 to (-90.44, -55.04, -4.17) mm, rotated rx -180 ry 0 rz -179 deg; joints [25.37, -71.975, 117.295, 33.699, -50.555, -22.962] to (-90.26, -55.49, -4.18) mm, rotated rx -180 ry 0 rz -179 deg; joints [25.384, -71.954, 117.267, 33.72, -50.555, -22.979]
  MoveL 966 to (-90.26, -80.89, -4.17) mm, rotated rx -180 ry 0 rz -179 deg; joints [26.401, -71.339, 116.409, 35.038, -50.759, -23.92]
  MoveL 967 to (-141.06, -80.89, -4.18) mm, rotated rx -180 ry 0 rz -179 deg; joints [27.394, -73.978, 120.035, 35.743, -51.966, -23.914]
  MoveL 968 to (-141.06, -30.09, -4.17) mm, rotated rx -180 ry 0 rz -179 deg; joints [25.284, -75.243, 121.725, 33.08, -51.493, -22.076]
  MoveL 969 to (-90.26, -30.09, -4.18) mm, rotated rx -180 ry 0 rz -179 deg; joints [24.351, -72.547, 118.086, 32.38, -50.349, -22.03]
  MoveL 970 to (-90.26, -55.49, -4.18) mm, rotated rx -180 ry 0 rz -179 deg; joints [25.384, -71.954, 117.267, 33.72, -50.555, -22.979]
  MoveC 971 to (-90.44, -55.94, -4.18) mm, rotated rx 180 ry 0 rz -179 deg; joints [25.406, -71.953, 117.265, 33.746, -50.563, -22.995] to (-90.89, -56.12, -4.17) mm, rotated rx -180 ry 0 rz -179 deg; joints [25.422, -71.972, 117.292, 33.761, -50.575, -23.002]
  MoveL 972 to (-91.53, -56.12, -4.17) mm, rotated rx -180 ry 0 rz -179 deg; joints [25.433, -72.006, 117.338, 33.769, -50.59, -23.001]
  MoveC 973 to (-91.98, -56.12, -3.99) mm, rotated rx -180 ry 0 rz -179 deg; joints [25.441, -72.037, 117.366, 33.78, -50.59, -23.01] to (-92.16, -56.12, -3.54) mm, rotated rx 180 ry 0 rz -179 deg; joints [25.445, -72.065, 117.367, 33.797, -50.569, -23.032]
  Set speed (500.0 mm/s)
  MoveL 974 to (-92.16, -56.12, 5) mm, rotated rx -180 ry 0 rz -179 deg; joints [25.445, -72.41, 117.126, 34.068, -50.083, -23.457]
  MoveL 975 to (-92.16, -54.85, 5) mm, rotated rx 180 ry 0 rz -179 deg; joints [25.394, -72.441, 117.168, 34.001, -50.072, -23.409]
  Set speed (25.4 mm/s)
  MoveL 976 to (-92.16, -54.85, 1.83) mm, rotated rx -180 ry 0 rz -179 deg; joints [25.394, -72.313, 117.258, 33.9, -50.253, -23.251]
  MoveL 977 to (-92.16, -54.85, -7.72) mm, rotated rx -180 ry 0 rz -179 deg; joints [25.394, -71.924, 117.524, 33.6, -50.797, -22.78]
  MoveC 978 to (-91.98, -54.85, -8.16) mm, rotated rx -180 ry 0 rz -179 deg; joints [25.39, -71.896, 117.523, 33.584, -50.818, -22.758] to (-91.53, -54.85, -8.35) mm, rotated rx 180 ry 0 rz -179 deg; joints [25.382, -71.865, 117.495, 33.573, -50.818, -22.749]
  Set speed (50.8 mm/s)
  MoveL 979 to (-90.89, -54.85, -8.35) mm, rotated rx -180 ry 0 rz -179 deg; joints [25.37, -71.832, 117.449, 33.565, -50.803, -22.75]
  MoveC 980 to (-90.44, -55.04, -8.35) mm, rotated rx 180 ry 0 rz -179 deg; joints [25.37, -71.804, 117.41, 33.569, -50.793, -22.757] to (-90.26, -55.49, -8.35) mm, rotated rx -180 ry 0 rz -179 deg; joints [25.384, -71.783, 117.382, 33.59, -50.793, -22.774]
  MoveL 981 to (-90.26, -80.89, -8.35) mm, rotated rx -180 ry 0 rz -179 deg; joints [26.401, -71.17, 116.524, 34.906, -50.992, -23.711]
  MoveL 982 to (-141.06, -80.89, -8.35) mm, rotated rx -180 ry 0 rz -179 deg; joints [27.394, -73.801, 120.152, 35.609, -52.205, -23.697]
  MoveL 983 to (-141.06, -30.09, -8.35) mm, rotated rx 180 ry 0 rz -179 deg; joints [25.284, -75.062, 121.843, 32.951, -51.743, -21.868]
  MoveL 984 to (-90.26, -30.09, -8.35) mm, rotated rx 180 ry 0 rz -179 deg; joints [24.351, -72.374, 118.201, 32.253, -50.592, -21.831]
  MoveL 985 to (-90.26, -55.49, -8.35) mm, rotated rx -180 ry 0 rz -179 deg; joints [25.384, -71.783, 117.382, 33.59, -50.793, -22.774]
  MoveC 986 to (-90.44, -55.94, -8.35) mm, rotated rx -180 ry 0 rz -179 deg; joints [25.406, -71.782, 117.38, 33.616, -50.801, -22.79] to (-90.89, -56.12, -8.35) mm, rotated rx 180 ry 0 rz -179 deg; joints [25.422, -71.801, 117.407, 33.631, -50.813, -22.797]
  MoveL 987 to (-91.53, -56.12, -8.35) mm, rotated rx 180 ry 0 rz -179 deg; joints [25.433, -71.835, 117.453, 33.639, -50.828, -22.796]
  MoveC 988 to (-91.98, -56.12, -8.16) mm, rotated rx -180 ry 0 rz -179 deg; joints [25.441, -71.866, 117.481, 33.65, -50.828, -22.805] to (-92.16, -56.12, -7.72) mm, rotated rx -180 ry 0 rz -179 deg; joints [25.445, -71.894, 117.482, 33.667, -50.807, -22.827]
  Set speed (500.0 mm/s)
  MoveL 989 to (-92.16, -56.12, 6) mm, rotated rx -180 ry 0 rz -179 deg; joints [25.445, -72.451, 117.098, 34.1, -50.026, -23.507]
  MoveL 990 to (-219.16, -54.85, 6) mm, rotated rx -180 ry 0 rz -179 deg; joints [27.949, -79.225, 125.953, 36.08, -52.734, -23.808]
  Set speed (25.4 mm/s)
  MoveL 991 to (-219.16, -54.85, -3.54) mm, rotated rx -180 ry 0 rz -179 deg; joints [27.949, -78.793, 126.239, 35.763, -53.315, -23.281]
  MoveC 992 to (-218.98, -54.85, -3.99) mm, rotated rx -180 ry 0 rz -179 deg; joints [27.945, -78.763, 126.24, 35.745, -53.339, -23.256] to (-218.53, -54.85, -4.17) mm, rotated rx -180 ry 0 rz -179 deg; joints [27.935, -78.731, 126.216, 35.73, -53.342, -23.243]
  Set speed (50.8 mm/s)
  MoveL 993 to (-217.89, -54.85, -4.17) mm, rotated rx -180 ry 0 rz -179 deg; joints [27.921, -78.697, 126.173, 35.718, -53.329, -23.24]
  MoveC 994 to (-217.44, -55.04, -4.18) mm, rotated rx -180 ry 0 rz -179 deg; joints [27.919, -78.668, 126.137, 35.719, -53.323, -23.244] to (-217.26, -55.49, -4.18) mm, rotated rx 180 ry 0 rz -179 deg; joints [27.934, -78.646, 126.11, 35.739, -53.324, -23.258]
  MoveL 995 to (-217.26, -80.89, -4.17) mm, rotated rx -180 ry 0 rz -179 deg; joints [29.024, -77.949, 125.231, 37.061, -53.616, -24.132]
  MoveL 996 to (-268.06, -80.89, -4.17) mm, rotated rx 180 ry 0 rz -179 deg; joints [30.218, -80.62, 128.542, 38.122, -54.614, -24.438]
  MoveL 997 to (-268.06, -30.09, -4.18) mm, rotated rx -180 ry 0 rz -179 deg; joints [27.953, -82.077, 130.283, 35.442, -53.935, -22.735]
  MoveL 998 to (-217.26, -30.09, -4.17) mm, rotated rx -180 ry 0 rz -179 deg; joints [26.823, -79.32, 126.95, 34.387, -53.029, -22.372]
  MoveL 999 to (-217.26, -55.49, -4.18) mm, rotated rx 180 ry 0 rz -179 deg; joints [27.934, -78.646, 126.11, 35.739, -53.324, -23.258]
  MoveC 1000 to (-217.44, -55.94, -4.17) mm, rotated rx -180 ry 0 rz -179 deg; joints [27.958, -78.644, 126.107, 35.766, -53.333, -23.275] to (-217.89, -56.12, -4.17) mm, rotated rx -180 ry 0 rz -179 deg; joints [27.976, -78.662, 126.13, 35.785, -53.344, -23.284]
  MoveL 1001 to (-218.53, -56.12, -4.18) mm, rotated rx -180 ry 0 rz -179 deg; joints [27.99, -78.696, 126.173, 35.797, -53.356, -23.287]
  MoveC 1002 to (-218.98, -56.12, -3.99) mm, rotated rx -180 ry 0 rz -179 deg; joints [28, -78.729, 126.197, 35.812, -53.354, -23.3] to (-219.16, -56.12, -3.54) mm, rotated rx 180 ry 0 rz -179 deg; joints [28.004, -78.759, 126.196, 35.83, -53.33, -23.325]
  Set speed (500.0 mm/s)
  MoveL 1003 to (-219.16, -56.12, 5) mm, rotated rx 180 ry 0 rz -179 deg; joints [28.004, -79.145, 125.941, 36.113, -52.811, -23.797]
  MoveL 1004 to (-219.16, -54.85, 5) mm, rotated rx 180 ry 0 rz -179 deg; joints [27.949, -79.18, 125.983, 36.046, -52.795, -23.753]
  Set speed (25.4 mm/s)
  MoveL 1005 to (-219.16, -54.85, 1.83) mm, rotated rx -180 ry 0 rz -179 deg; joints [27.949, -79.037, 126.079, 35.94, -52.988, -23.577]
  MoveL 1006 to (-219.16, -54.85, -7.72) mm, rotated rx 180 ry 0 rz -179 deg; joints [27.949, -78.602, 126.362, 35.627, -53.57, -23.053]
  MoveC 1007 to (-218.98, -54.85, -8.16) mm, rotated rx 180 ry 0 rz -179 deg; joints [27.945, -78.571, 126.363, 35.609, -53.594, -23.028] to (-218.53, -54.85, -8.35) mm, rotated rx -180 ry 0 rz -179 deg; joints [27.935, -78.539, 126.338, 35.594, -53.597, -23.015]
  Set speed (50.8 mm/s)
  MoveL 1008 to (-217.89, -54.85, -8.35) mm, rotated rx 180 ry 0 rz -179 deg; joints [27.921, -78.505, 126.296, 35.582, -53.584, -23.012]
  MoveC 1009 to (-217.44, -55.04, -8.35) mm, rotated rx -180 ry 0 rz -179 deg; joints [27.919, -78.477, 126.26, 35.583, -53.578, -23.016] to (-217.26, -55.49, -8.35) mm, rotated rx -180 ry 0 rz -179 deg; joints [27.934, -78.455, 126.232, 35.603, -53.579, -23.031]
  MoveL 1010 to (-217.26, -80.89, -8.35) mm, rotated rx -180 ry 0 rz -179 deg; joints [29.024, -77.76, 125.353, 36.924, -53.864, -23.9]
  MoveL 1011 to (-268.06, -80.89, -8.35) mm, rotated rx -180 ry 0 rz -179 deg; joints [30.218, -80.422, 128.667, 37.981, -54.868, -24.194]
  MoveL 1012 to (-268.06, -30.09, -8.35) mm, rotated rx 180 ry 0 rz -179 deg; joints [27.953, -81.875, 130.411, 35.304, -54.204, -22.499]
  MoveL 1013 to (-217.26, -30.09, -8.35) mm, rotated rx -180 ry 0 rz -179 deg; joints [26.823, -79.127, 127.073, 34.254, -53.29, -22.149]
  MoveL 1014 to (-217.26, -55.49, -8.35) mm, rotated rx -180 ry 0 rz -179 deg; joints [27.934, -78.455, 126.232, 35.603, -53.579, -23.031]
  MoveC 1015 to (-217.44, -55.94, -8.35) mm, rotated rx -180 ry 0 rz -179 deg; joints [27.958, -78.452, 126.229, 35.63, -53.588, -23.047] to (-217.89, -56.12, -8.35) mm, rotated rx 180 ry 0 rz -179 deg; joints [27.976, -78.471, 126.253, 35.649, -53.599, -23.056]
  MoveL 1016 to (-218.53, -56.12, -8.35) mm, rotated rx -180 ry 0 rz -179 deg; joints [27.99, -78.505, 126.295, 35.661, -53.611, -23.059]
  MoveC 1017 to (-218.98, -56.12, -8.16) mm, rotated rx -180 ry 0 rz -179 deg; joints [28, -78.537, 126.32, 35.676, -53.609, -23.071] to (-219.16, -56.12, -7.72) mm, rotated rx 180 ry 0 rz -179 deg; joints [28.004, -78.568, 126.319, 35.694, -53.585, -23.097]
  Set speed (500.0 mm/s)
  MoveL 1018 to (-219.16, -56.12, 6) mm, rotated rx 180 ry 0 rz -179 deg; joints [28.004, -79.19, 125.91, 36.147, -52.75, -23.853]
  MoveL 1019 to (-346.16, -54.85, 6) mm, rotated rx -180 ry 0 rz -179 deg; joints [31.047, -86.142, 133.999, 39.072, -54.911, -25.018]
  Set speed (25.4 mm/s)
  MoveL 1020 to (-346.16, -54.85, -3.54) mm, rotated rx -180 ry 0 rz -179 deg; joints [31.047, -85.661, 134.309, 38.727, -55.526, -24.414]
  MoveC 1021 to (-345.98, -54.85, -3.99) mm, rotated rx -180 ry 0 rz -179 deg; joints [31.042, -85.628, 134.313, 38.705, -55.552, -24.383] to (-345.53, -54.85, -4.17) mm, rotated rx -180 ry 0 rz -179 deg; joints [31.03, -85.593, 134.291, 38.687, -55.557, -24.366]
  Set speed (50.8 mm/s)
  MoveL 1022 to (-344.89, -54.85, -4.17) mm, rotated rx -180 ry 0 rz -179 deg; joints [31.013, -85.558, 134.253, 38.669, -55.548, -24.358]
  MoveC 1023 to (-344.44, -55.04, -4.17) mm, rotated rx -180 ry 0 rz -179 deg; joints [31.009, -85.528, 134.219, 38.667, -55.544, -24.358] to (-344.26, -55.49, -4.17) mm, rotated rx -180 ry 0 rz -179 deg; joints [31.025, -85.503, 134.192, 38.685, -55.548, -24.37]
  MoveL 1024 to (-344.26, -80.89, -4.18) mm, rotated rx 180 ry 0 rz -179 deg; joints [32.192, -84.684, 133.282, 40.007, -55.966, -25.161]
  MoveL 1025 to (-395.06, -80.89, -4.18) mm, rotated rx -180 ry 0 rz -179 deg; joints [33.646, -87.446, 136.291, 41.476, -56.78, -25.84]
  MoveL 1026 to (-395.06, -30.09, -4.17) mm, rotated rx -180 ry 0 rz -179 deg; joints [31.22, -89.192, 138.104, 38.804, -55.803, -24.321]
  MoveL 1027 to (-344.26, -30.09, -4.18) mm, rotated rx -180 ry 0 rz -179 deg; joints [29.83, -86.301, 135.064, 37.326, -55.122, -23.559]
  MoveL 1028 to (-344.26, -55.49, -4.17) mm, rotated rx -180 ry 0 rz -179 deg; joints [31.025, -85.503, 134.192, 38.685, -55.548, -24.37]
  MoveC 1029 to (-344.44, -55.94, -4.18) mm, rotated rx 180 ry 0 rz -179 deg; joints [31.051, -85.499, 134.187, 38.714, -55.559, -24.386] to (-344.89, -56.12, -4.18) mm, rotated rx -180 ry 0 rz -179 deg; joints [31.072, -85.518, 134.208, 38.736, -55.569, -24.398]
  MoveL 1030 to (-345.53, -56.12, -4.18) mm, rotated rx -180 ry 0 rz -179 deg; joints [31.089, -85.553, 134.247, 38.754, -55.579, -24.406]
  MoveC 1031 to (-345.98, -56.12, -3.99) mm, rotated rx -180 ry 0 rz -179 deg; joints [31.101, -85.587, 134.268, 38.773, -55.574, -24.423] to (-346.16, -56.12, -3.54) mm, rotated rx -180 ry 0 rz -179 deg; joints [31.106, -85.62, 134.265, 38.794, -55.547, -24.454]
  Set speed (500.0 mm/s)
  MoveL 1032 to (-346.16, -56.12, 5) mm, rotated rx 180 ry 0 rz -179 deg; joints [31.106, -86.051, 133.988, 39.102, -54.997, -24.995]
  MoveL 1033 to (-346.16, -54.85, 5) mm, rotated rx 180 ry 0 rz -179 deg; joints [31.047, -86.092, 134.032, 39.035, -54.975, -24.955]
  Set speed (25.4 mm/s)
  MoveL 1034 to (-346.16, -54.85, 1.82) mm, rotated rx -180 ry 0 rz -179 deg; joints [31.047, -85.932, 134.136, 38.919, -55.179, -24.753]
  MoveL 1035 to (-346.16, -54.85, -7.72) mm, rotated rx 180 ry 0 rz -179 deg; joints [31.047, -85.447, 134.443, 38.579, -55.797, -24.151]
  MoveC 1036 to (-345.98, -54.85, -8.16) mm, rotated rx -180 ry 0 rz -179 deg; joints [31.042, -85.414, 134.446, 38.558, -55.823, -24.121] to (-345.53, -54.85, -8.35) mm, rotated rx -180 ry 0 rz -179 deg; joints [31.03, -85.38, 134.424, 38.539, -55.828, -24.104]
  Set speed (50.8 mm/s)
  MoveL 1037 to (-344.89, -54.85, -8.35) mm, rotated rx -180 ry 0 rz -179 deg; joints [31.013, -85.345, 134.386, 38.522, -55.819, -24.096]
  MoveC 1038 to (-344.44, -55.04, -8.35) mm, rotated rx -180 ry 0 rz -179 deg; joints [31.009, -85.314, 134.352, 38.519, -55.815, -24.096] to (-344.26, -55.49, -8.35) mm, rotated rx 180 ry 0 rz -179 deg; joints [31.025, -85.29, 134.325, 38.538, -55.819, -24.108]
  MoveL 1039 to (-344.26, -80.89, -8.35) mm, rotated rx -180 ry 0 rz -179 deg; joints [32.192, -84.474, 133.413, 39.859, -56.229, -24.897]
  MoveL 1040 to (-395.06, -80.89, -8.35) mm, rotated rx -180 ry 0 rz -179 deg; joints [33.646, -87.226, 136.427, 41.322, -57.048, -25.559]
  MoveL 1041 to (-395.06, -30.09, -8.35) mm, rotated rx -180 ry 0 rz -179 deg; joints [31.22, -88.966, 138.244, 38.65, -56.088, -24.046]
  MoveL 1042 to (-344.26, -30.09, -8.35) mm, rotated rx -180 ry 0 rz -179 deg; joints [29.83, -86.085, 135.198, 37.179, -55.401, -23.301]
  MoveL 1043 to (-344.26, -55.49, -8.35) mm, rotated rx 180 ry 0 rz -179 deg; joints [31.025, -85.29, 134.325, 38.538, -55.819, -24.108]
  MoveC 1044 to (-344.44, -55.94, -8.35) mm, rotated rx -180 ry 0 rz -179 deg; joints [31.051, -85.286, 134.32, 38.567, -55.829, -24.124] to (-344.89, -56.12, -8.35) mm, rotated rx -180 ry 0 rz -179 deg; joints [31.072, -85.305, 134.341, 38.589, -55.839, -24.136]
  MoveL 1045 to (-345.53, -56.12, -8.35) mm, rotated rx 180 ry 0 rz -179 deg; joints [31.089, -85.339, 134.38, 38.606, -55.849, -24.144]
  MoveC 1046 to (-345.98, -56.12, -8.16) mm, rotated rx 180 ry 0 rz -179 deg; joints [31.101, -85.374, 134.401, 38.625, -55.844, -24.161] to (-346.16, -56.12, -7.72) mm, rotated rx -180 ry 0 rz -179 deg; joints [31.106, -85.407, 134.398, 38.646, -55.818, -24.191]
  Set speed (500.0 mm/s)
  MoveL 1047 to (-346.16, -56.12, 15) mm, rotated rx -180 ry 0 rz -179 deg; joints [31.106, -86.545, 133.655, 39.473, -54.357, -25.636]
  Print: /'2D Contour1'
  Set speed (500.0 mm/s)
  MoveL 1048 to (-12.15, 15.92, 15) mm, rotated rx -180 ry 0 rz -179 deg; joints [21.216, -70.092, 113.064, 29.661, -46.992, -21.229]
  MoveL 1049 to (-12.15, 15.92, 6) mm, rotated rx -180 ry 0 rz -179 deg; joints [21.216, -69.75, 113.32, 29.389, -47.512, -20.828]
  Set speed (25.4 mm/s)
  MoveL 1050 to (-12.15, 15.92, -4.36) mm, rotated rx 180 ry 0 rz -179 deg; joints [21.216, -69.35, 113.606, 29.085, -48.112, -20.375]
  MoveC 1051 to (-12.34, 15.92, -4.81) mm, rotated rx -180 ry 0 rz -179 deg; joints [21.218, -69.342, 113.633, 29.074, -48.142, -20.355] to (-12.79, 15.92, -5) mm, rotated rx -180 ry 0 rz -179 deg; joints [21.225, -69.359, 113.673, 29.072, -48.165, -20.346]
  Set speed (50.8 mm/s)
  MoveL 1052 to (-13.42, 15.92, -5) mm, rotated rx 180 ry 0 rz -179 deg; joints [21.235, -69.393, 113.722, 29.077, -48.181, -20.344]
  MoveC 1053 to (-13.87, 16.1, -5) mm, rotated rx -180 ry 0 rz -179 deg; joints [21.234, -69.421, 113.762, 29.071, -48.191, -20.335] to (-14.06, 16.55, -5) mm, rotated rx -180 ry 0 rz -179 deg; joints [21.218, -69.44, 113.789, 29.048, -48.193, -20.317]
  MoveL 1054 to (-14.06, 168.95, -5) mm, rotated rx -180 ry 0 rz -179 deg; joints [14.861, -72.009, 117.412, 20.438, -47.264, -14.192]
  MoveL 1055 to (-39.46, 168.95, -5) mm, rotated rx -180 ry 0 rz -179 deg; joints [15.136, -73.431, 119.365, 20.629, -47.828, -14.184]
  MoveC 1056 to (-52.16, 156.25, -5) mm, rotated rx 180 ry 0 rz -179 deg; joints [15.839, -73.96, 120.081, 21.484, -48.178, -14.706] to (-64.86, 168.95, -5) mm, rotated rx -180 ry 0 rz -179 deg; joints [15.422, -74.86, 121.287, 20.845, -48.36, -14.198]
  MoveL 1057 to (-90.26, 168.95, -5) mm, rotated rx 180 ry 0 rz -179 deg; joints [15.72, -76.296, 123.179, 21.086, -48.858, -14.235]
  MoveL 1058 to (-166.46, 168.95, -5) mm, rotated rx -180 ry 0 rz -179 deg; joints [16.69, -80.674, 128.679, 21.97, -50.143, -14.496]
  MoveC 1059 to (-179.16, 156.25, -5) mm, rotated rx 180 ry 0 rz -179 deg; joints [17.48, -81.201, 129.314, 22.929, -50.444, -15.077] to (-191.86, 168.95, -5) mm, rotated rx -180 ry 0 rz -179 deg; joints [17.041, -82.163, 130.457, 22.322, -50.498, -14.637]
  MoveL 1060 to (-293.46, 168.95, -5) mm, rotated rx -180 ry 0 rz -179 deg; joints [18.615, -88.335, 137.296, 24.064, -51.521, -15.529]
  MoveC 1061 to (-306.16, 156.25, -5) mm, rotated rx -180 ry 0 rz -179 deg; joints [19.516, -88.873, 137.851, 25.163, -51.783, -16.205] to (-318.86, 168.95, -5) mm, rotated rx 180 ry 0 rz -179 deg; joints [19.056, -89.946, 138.939, 24.595, -51.669, -15.849]
  MoveL 1062 to (-395.06, 168.95, -5) mm, rotated rx -180 ry 0 rz -179 deg; joints [20.517, -94.99, 143.698, 26.476, -51.827, -17.11]
  MoveL 1063 to (-420.46, 168.95, -5) mm, rotated rx -180 ry 0 rz -179 deg; joints [21.056, -96.755, 145.227, 27.214, -51.778, -17.65]
  MoveC 1064 to (-433.16, 156.25, -5) mm, rotated rx 180 ry 0 rz -179 deg; joints [22.099, -97.314, 145.697, 28.507, -52.022, -18.48] to (-445.86, 168.95, -5) mm, rotated rx 180 ry 0 rz -179 deg; joints [21.624, -98.567, 146.725, 28.018, -51.674, -18.262]
  MoveL 1065 to (-471.26, 168.95, -5) mm, rotated rx 180 ry 0 rz -179 deg; joints [22.224, -100.432, 148.192, 28.894, -51.516, -18.954]
  MoveL 1066 to (-471.26, 16.55, -5) mm, rotated rx 180 ry 0 rz -179 deg; joints [31.098, -95.373, 144.036, 38.777, -55.558, -24.435]
  MoveL 1067 to (-14.06, 16.55, -5) mm, rotated rx -180 ry 0 rz -179 deg; joints [21.218, -69.44, 113.789, 29.048, -48.193, -20.317]
  MoveC 1068 to (-13.61, 16.36, -5) mm, rotated rx -180 ry 0 rz -179 deg; joints [21.219, -69.412, 113.749, 29.055, -48.183, -20.326] to (-13.42, 15.92, -5) mm, rotated rx 180 ry 0 rz -179 deg; joints [21.235, -69.393, 113.722, 29.077, -48.181, -20.344]
  MoveL 1069 to (-13.42, 15.28, -5) mm, rotated rx -180 ry 0 rz -179 deg; joints [21.26, -69.381, 113.704, 29.112, -48.185, -20.369]
  MoveC 1070 to (-13.42, 14.83, -4.81) mm, rotated rx 180 ry 0 rz -179 deg; joints [21.278, -69.379, 113.686, 29.142, -48.177, -20.394] to (-13.42, 14.65, -4.37) mm, rotated rx -180 ry 0 rz -179 deg; joints [21.286, -69.393, 113.668, 29.165, -48.152, -20.421]
  Set speed (500.0 mm/s)
  MoveL 1071 to (-13.42, 14.65, 5) mm, rotated rx -180 ry 0 rz -179 deg; joints [21.286, -69.755, 113.41, 29.439, -47.611, -20.831]
  MoveL 1072 to (-12.15, 15.92, 5) mm, rotated rx 180 ry 0 rz -179 deg; joints [21.216, -69.712, 113.348, 29.359, -47.57, -20.784]
  Set speed (25.4 mm/s)
  MoveL 1073 to (-12.15, 15.92, 1) mm, rotated rx -180 ry 0 rz -179 deg; joints [21.216, -69.558, 113.459, 29.241, -47.801, -20.608]
  MoveL 1074 to (-12.15, 15.92, -7.72) mm, rotated rx 180 ry 0 rz -179 deg; joints [21.216, -69.219, 113.697, 28.989, -48.306, -20.23]
  MoveC 1075 to (-12.34, 15.92, -8.16) mm, rotated rx -180 ry 0 rz -179 deg; joints [21.218, -69.211, 113.724, 28.977, -48.336, -20.211] to (-12.79, 15.92, -8.35) mm, rotated rx -180 ry 0 rz -179 deg; joints [21.225, -69.228, 113.763, 28.976, -48.359, -20.201]
  Set speed (50.8 mm/s)
  MoveL 1076 to (-13.42, 15.92, -8.35) mm, rotated rx 180 ry 0 rz -179 deg; joints [21.235, -69.262, 113.812, 28.981, -48.375, -20.199]
  MoveC 1077 to (-13.87, 16.1, -8.35) mm, rotated rx 180 ry 0 rz -179 deg; joints [21.234, -69.29, 113.852, 28.975, -48.386, -20.191] to (-14.06, 16.55, -8.35) mm, rotated rx 180 ry 0 rz -179 deg; joints [21.218, -69.309, 113.879, 28.952, -48.387, -20.173]
  MoveL 1078 to (-14.06, 168.95, -8.35) mm, rotated rx -180 ry 0 rz -179 deg; joints [14.861, -71.872, 117.504, 20.364, -47.479, -14.083]
  MoveL 1079 to (-39.46, 168.95, -8.35) mm, rotated rx -180 ry 0 rz -179 deg; joints [15.136, -73.291, 119.459, 20.555, -48.047, -14.073]
  MoveC 1080 to (-52.16, 156.25, -8.35) mm, rotated rx 180 ry 0 rz -179 deg; joints [15.839, -73.818, 120.175, 21.407, -48.397, -14.59] to (-64.86, 168.95, -8.35) mm, rotated rx -180 ry 0 rz -179 deg; joints [15.422, -74.716, 121.382, 20.77, -48.583, -14.085]
  MoveL 1081 to (-90.26, 168.95, -8.35) mm, rotated rx -180 ry 0 rz -179 deg; joints [15.72, -76.149, 123.275, 21.01, -49.085, -14.119]
  MoveL 1082 to (-166.46, 168.95, -8.35) mm, rotated rx -180 ry 0 rz -179 deg; joints [16.69, -80.515, 128.78, 21.889, -50.383, -14.37]
  MoveC 1083 to (-179.16, 156.25, -8.35) mm, rotated rx -180 ry 0 rz -179 deg; joints [17.48, -81.041, 129.415, 22.845, -50.684, -14.945] to (-191.86, 168.95, -8.35) mm, rotated rx -180 ry 0 rz -179 deg; joints [17.041, -82.001, 130.559, 22.239, -50.743, -14.507]
  MoveL 1084 to (-293.46, 168.95, -8.35) mm, rotated rx -180 ry 0 rz -179 deg; joints [18.615, -88.156, 137.407, 23.97, -51.786, -15.378]
  MoveC 1085 to (-306.16, 156.25, -8.35) mm, rotated rx 180 ry 0 rz -179 deg; joints [19.516, -88.693, 137.963, 25.066, -52.047, -16.048] to (-318.86, 168.95, -8.35) mm, rotated rx -180 ry 0 rz -179 deg; joints [19.056, -89.763, 139.052, 24.498, -51.939, -15.692]
  MoveL 1086 to (-395.06, 168.95, -8.35) mm, rotated rx -180 ry 0 rz -179 deg; joints [20.517, -94.794, 143.82, 26.366, -52.112, -16.93]
  MoveL 1087 to (-420.46, 168.95, -8.35) mm, rotated rx 180 ry 0 rz -179 deg; joints [21.056, -96.554, 145.352, 27.098, -52.067, -17.461]
  MoveC 1088 to (-433.16, 156.25, -8.35) mm, rotated rx 180 ry 0 rz -179 deg; joints [22.099, -97.112, 145.823, 28.386, -52.31, -18.282] to (-445.86, 168.95, -8.35) mm, rotated rx -180 ry 0 rz -179 deg; joints [21.624, -98.363, 146.854, 27.895, -51.968, -18.063]
  MoveL 1089 to (-471.26, 168.95, -8.35) mm, rotated rx 180 ry 0 rz -179 deg; joints [22.224, -100.223, 148.324, 28.764, -51.814, -18.745]
  MoveL 1090 to (-471.26, 16.55, -8.35) mm, rotated rx -180 ry 0 rz -179 deg; joints [31.098, -95.176, 144.159, 38.641, -55.808, -24.193]
  MoveL 1091 to (-14.06, 16.55, -8.35) mm, rotated rx 180 ry 0 rz -179 deg; joints [21.218, -69.309, 113.879, 28.952, -48.387, -20.173]
  MoveC 1092 to (-13.61, 16.36, -8.35) mm, rotated rx -180 ry 0 rz -179 deg; joints [21.219, -69.281, 113.84, 28.959, -48.377, -20.181] to (-13.42, 15.92, -8.35) mm, rotated rx 180 ry 0 rz -179 deg; joints [21.235, -69.262, 113.812, 28.981, -48.375, -20.199]
  MoveL 1093 to (-13.42, 15.28, -8.35) mm, rotated rx 180 ry 0 rz -179 deg; joints [21.26, -69.25, 113.794, 29.016, -48.379, -20.224]
  MoveC 1094 to (-13.42, 14.83, -8.16) mm, rotated rx -180 ry 0 rz -179 deg; joints [21.278, -69.248, 113.777, 29.045, -48.371, -20.25] to (-13.42, 14.65, -7.72) mm, rotated rx -180 ry 0 rz -179 deg; joints [21.286, -69.262, 113.759, 29.068, -48.346, -20.276]
  Set speed (500.0 mm/s)
  MoveL 1095 to (-13.42, 14.65, 6) mm, rotated rx 180 ry 0 rz -179 deg; joints [21.286, -69.794, 113.382, 29.469, -47.553, -20.875]
  MoveL 1096 to (18.41, 14.65, 6) mm, rotated rx 180 ry 0 rz -179 deg; joints [20.823, -68.068, 110.9, 29.224, -46.729, -20.98]
  Set speed (25.4 mm/s)
  MoveL 1097 to (18.41, 14.65, -4.37) mm, rotated rx -180 ry 0 rz -179 deg; joints [20.823, -67.679, 111.184, 28.919, -47.317, -20.533]
  MoveC 1098 to (18.41, 14.83, -4.81) mm, rotated rx 180 ry 0 rz -179 deg; joints [20.816, -67.666, 111.201, 28.896, -47.341, -20.507] to (18.41, 15.28, -5) mm, rotated rx -180 ry 0 rz -179 deg; joints [20.798, -67.668, 111.219, 28.867, -47.349, -20.481]
  Set speed (50.8 mm/s)
  MoveL 1099 to (18.41, 15.92, -5) mm, rotated rx -180 ry 0 rz -179 deg; joints [20.773, -67.68, 111.237, 28.832, -47.345, -20.455]
  MoveC 1100 to (18.6, 16.36, -5) mm, rotated rx 180 ry 0 rz -179 deg; joints [20.753, -67.679, 111.235, 28.806, -47.338, -20.438] to (19.04, 16.55, -5) mm, rotated rx -180 ry 0 rz -179 deg; joints [20.739, -67.658, 111.205, 28.793, -47.325, -20.433]
  MoveL 1101 to (39.46, 16.55, -5) mm, rotated rx -180 ry 0 rz -179 deg; joints [20.454, -66.556, 109.58, 28.663, -46.766, -20.528]
  MoveL 1102 to (471.26, 16.55, -5) mm, rotated rx -180 ry 0 rz -179 deg; joints [15.87, -40.376, 66.028, 33.293, -29.879, -29.658]
  MoveL 1103 to (471.26, 168.95, -5) mm, rotated rx -180 ry 0 rz -179 deg; joints [11.087, -42.88, 70.526, 22.896, -29.623, -20.16]
  MoveL 1104 to (445.86, 168.95, -5) mm, rotated rx -180 ry 0 rz -179 deg; joints [11.234, -44.69, 73.741, 22.246, -30.97, -19.326]
  MoveC 1105 to (433.16, 156.25, -5) mm, rotated rx -180 ry 0 rz -179 deg; joints [11.722, -45.408, 75.008, 22.786, -31.64, -19.679] to (420.46, 168.95, -5) mm, rotated rx -180 ry 0 rz -179 deg; joints [11.384, -46.436, 76.813, 21.711, -32.248, -18.611]
  MoveL 1106 to (395.06, 168.95, -5) mm, rotated rx -180 ry 0 rz -179 deg; joints [11.539, -48.129, 79.761, 21.271, -33.465, -17.992]
  MoveL 1107 to (318.86, 168.95, -5) mm, rotated rx 180 ry 0 rz -179 deg; joints [12.033, -52.955, 87.995, 20.369, -36.797, -16.557]
  MoveC 1108 to (306.16, 156.25, -5) mm, rotated rx -180 ry 0 rz -179 deg; joints [12.565, -53.575, 89.034, 21.017, -37.342, -16.985] to (293.46, 168.95, -5) mm, rotated rx -180 ry 0 rz -179 deg; joints [12.208, -54.498, 90.571, 20.176, -37.815, -16.187]
  MoveL 1109 to (191.86, 168.95, -5) mm, rotated rx -180 ry 0 rz -179 deg; joints [12.967, -60.45, 100.217, 19.797, -41.492, -15.089]
  MoveC 1110 to (179.16, 156.25, -5) mm, rotated rx -180 ry 0 rz -179 deg; joints [13.549, -61.017, 101.112, 20.514, -41.953, -15.55] to (166.46, 168.95, -5) mm, rotated rx -180 ry 0 rz -179 deg; joints [13.172, -61.898, 102.49, 19.783, -42.321, -14.893]
  MoveL 1111 to (90.26, 168.95, -5) mm, rotated rx -180 ry 0 rz -179 deg; joints [13.833, -66.187, 109.031, 19.906, -44.607, -14.456]
  MoveL 1112 to (64.86, 168.95, -5) mm, rotated rx -180 ry 0 rz -179 deg; joints [14.069, -67.606, 111.129, 19.998, -45.304, -14.358]
  MoveC 1113 to (61.14, 159.97, -5) mm, rotated rx 180 ry 0 rz -179 deg; joints [14.471, -67.695, 111.26, 20.53, -45.444, -14.721] to (52.16, 156.25, -5) mm, rotated rx 180 ry 0 rz -179 deg; joints [14.712, -68.145, 111.917, 20.785, -45.699, -14.847]
  MoveL 1114 to (52.16, 156.25, -5) mm, rotated rx -180 ry 0 rz -179 deg; joints [14.712, -68.145, 111.917, 20.785, -45.699, -14.847]
  MoveC 1115 to (43.18, 159.97, -5) mm, rotated rx -180 ry 0 rz -179 deg; joints [14.649, -68.695, 112.716, 20.614, -45.916, -14.665] to (39.46, 168.95, -5) mm, rotated rx -180 ry 0 rz -179 deg; joints [14.314, -69.023, 113.188, 20.114, -45.968, -14.281]
  MoveL 1116 to (14.06, 168.95, -5) mm, rotated rx -180 ry 0 rz -179 deg; joints [14.568, -70.439, 115.212, 20.254, -46.601, -14.227]
  MoveL 1117 to (14.06, 16.55, -5) mm, rotated rx -180 ry 0 rz -179 deg; joints [20.81, -67.927, 111.598, 28.828, -47.458, -20.412]
  MoveL 1118 to (19.04, 16.55, -5) mm, rotated rx -180 ry 0 rz -179 deg; joints [20.739, -67.658, 111.205, 28.793, -47.325, -20.433]
  MoveC 1119 to (19.49, 16.36, -5) mm, rotated rx -180 ry 0 rz -179 deg; joints [20.74, -67.63, 111.164, 28.8, -47.314, -20.442] to (19.68, 15.92, -5) mm, rotated rx -180 ry 0 rz -179 deg; joints [20.755, -67.611, 111.137, 28.823, -47.311, -20.461]
  MoveL 1120 to (19.68, 15.28, -5) mm, rotated rx -180 ry 0 rz -179 deg; joints [20.78, -67.599, 111.119, 28.858, -47.315, -20.486]
  MoveC 1121 to (19.68, 14.83, -4.81) mm, rotated rx 180 ry 0 rz -179 deg; joints [20.798, -67.597, 111.101, 28.888, -47.307, -20.512] to (19.68, 14.65, -4.37) mm, rotated rx -180 ry 0 rz -179 deg; joints [20.805, -67.611, 111.083, 28.911, -47.283, -20.539]
  Set speed (500.0 mm/s)
  MoveL 1122 to (19.68, 14.65, 5) mm, rotated rx -180 ry 0 rz -179 deg; joints [20.805, -67.962, 110.827, 29.186, -46.751, -20.942]
  MoveL 1123 to (18.41, 14.65, 5) mm, rotated rx 180 ry 0 rz -179 deg; joints [20.823, -68.031, 110.928, 29.194, -46.785, -20.937]
  Set speed (25.4 mm/s)
  MoveL 1124 to (18.41, 14.65, 1) mm, rotated rx -180 ry 0 rz -179 deg; joints [20.823, -67.882, 111.038, 29.076, -47.012, -20.763]
  MoveL 1125 to (18.41, 14.65, -7.72) mm, rotated rx -180 ry 0 rz -179 deg; joints [20.823, -67.552, 111.274, 28.823, -47.507, -20.391]
  MoveC 1126 to (18.41, 14.83, -8.16) mm, rotated rx 180 ry 0 rz -179 deg; joints [20.816, -67.538, 111.291, 28.8, -47.532, -20.364] to (18.41, 15.28, -8.35) mm, rotated rx -180 ry 0 rz -179 deg; joints [20.798, -67.54, 111.309, 28.77, -47.539, -20.339]
  Set speed (50.8 mm/s)
  MoveL 1127 to (18.41, 15.92, -8.35) mm, rotated rx -180 ry 0 rz -179 deg; joints [20.773, -67.552, 111.327, 28.736, -47.536, -20.313]
  MoveC 1128 to (18.6, 16.36, -8.35) mm, rotated rx 180 ry 0 rz -179 deg; joints [20.753, -67.551, 111.325, 28.71, -47.528, -20.296] to (19.05, 16.55, -8.35) mm, rotated rx -180 ry 0 rz -179 deg; joints [20.739, -67.53, 111.295, 28.697, -47.515, -20.291]
  MoveL 1129 to (39.46, 16.55, -8.35) mm, rotated rx -180 ry 0 rz -179 deg; joints [20.454, -66.431, 109.669, 28.567, -46.954, -20.387]
  MoveL 1130 to (471.26, 16.55, -8.35) mm, rotated rx -180 ry 0 rz -179 deg; joints [15.87, -40.302, 66.135, 33.122, -30.03, -29.461]
  MoveL 1131 to (471.26, 168.95, -8.35) mm, rotated rx 180 ry 0 rz -179 deg; joints [11.087, -42.801, 70.627, 22.773, -29.789, -20.019]
  MoveL 1132 to (445.86, 168.95, -8.35) mm, rotated rx -180 ry 0 rz -179 deg; joints [11.234, -44.607, 73.839, 22.132, -31.137, -19.194]
